// TwinCAT 3 PLC project LoadPCBAProject
// ProgramVersion: 3.1.4023.0
// libraries:
//   GreatechTemplate, * (Greatech)
//   Tc2_Standard, * (Beckhoff Automation GmbH)
//   Tc2_System, * (Beckhoff Automation GmbH)
//   Tc2_Utilities, * (Beckhoff Automation GmbH)
//   Tc3_Module, * (Beckhoff Automation GmbH)
// project tree:
//   DUTs/ ST_BarcodeScanner.TcDUT, ST_ModulePerformance.TcDUT, ST_OEETime.TcDUT, ST_Position.TcDUT, ST_ScaraCurrentPos.TcDUT, ST_ScaraRobot.TcDUT, ST_ScaraRobotCmd.TcDUT, ST_VisionRecipe.TcDUT
//   GVLs/ DeviceMapping.TcGVL, G_Auto.TcGVL, G_Error.TcGVL, G_Home.TcGVL, G_IO.TcGVL, G_MachineControl.TcGVL, G_Manual.TcGVL, G_Recipe.TcGVL, G_Robot.TcGVL, G_Safety.TcGVL, G_Scanner.TcGVL, G_Values.TcGVL, G_Vision.TcGVL
//   / PlcTask.TcTTO
//   POUs/Function Block/ FB_CognexBarcodeScanner.TcPOU, FB_OEETime.TcPOU, FB_RealToBytes.TcPOU
//   POUs/Function/ F_BytesToWord.TcPOU, F_ReadRobotPosition.TcPOU
//   POUs/General/ DoorLock.TcPOU, ErrorHandle.TcPOU, Initialize.TcPOU, MAIN.TcPOU, NewLotEndLot.TcPOU
//   POUs/General/Mapping/ Mapping_EIP.TcPOU, Mapping_IO.TcPOU
//   POUs/ POU_TestGitHub.TcPOU
//   POUs/Station/ST00_Conveyor/ ST00_ChangeRecipe.TcPOU, ST00_Cylinder.TcPOU, ST00_Sequence.TcPOU
//   POUs/Station/ST10_BarcodeScanner/ ST10_BarcodeScanner.TcPOU, ST10_Sequence.TcPOU
//   POUs/Station/ST20_PickNPlace/Robot/ ST20_RobotManualControl.TcPOU, ST20_RobotSequence.TcPOU, ST20_VisionManualControl.TcPOU
//   POUs/Station/ST20_PickNPlace/ ST20_ChangeRecipe.TcPOU, ST20_Home.TcPOU, ST20_Sequence.TcPOU
//   POUs/Station/ST20_PickNPlace/TrayLoader/ ST20_TraySequence.TcPOU, ST20_BarcodeScanner.TcPOU
// real-time tasks:
//   TASK PlcTask: cycle T#10ms, priority 20, ADS port 350

CONFIGURATION LoadPCBAProject
    RESOURCE PLC ON TwinCAT3
        TASK PlcTask(INTERVAL := T#10ms, PRIORITY := 20);
        PROGRAM MAIN WITH PlcTask : MAIN;
    END_RESOURCE
END_CONFIGURATION

// ---- DUTs/ST_BarcodeScanner.TcDUT
TYPE ST_BarcodeScanner :
STRUCT
	In_TriggerReady			: BOOL;
	In_TriggerAck			: BOOL;
	In_Acquiring			: BOOL;
	In_MissedAcq			: BOOL;
	In_noname0_arrBIT_0		: BOOL;
	In_noname0_arrBIT_1		: BOOL;
	In_noname0_arrBIT_2		: BOOL;
	In_noname0_arrBIT_3		: BOOL;
	In_Decoding				: BOOL;
	In_DecodeComplete		: BOOL;
	In_ResultsBufferOverrun : BOOL;
	In_ResultAvailable		: BOOL;
	In_noname1_arrBIT_0		: BOOL;
	In_noname1_arrBIT_1		: BOOL;
	In_noname1_arrBIT_2		: BOOL;
	In_GeneralFault			: BOOL;
	In_SoftEventAck0		: BOOL;
	In_SoftEventAck1		: BOOL;
	In_SoftEventAck2		: BOOL;
	In_SoftEventAck3		: BOOL;
	In_SoftEventAck4		: BOOL;
	In_SoftEventAck5		: BOOL;
	In_SoftEventAck6		: BOOL;
	In_SoftEventAck7		: BOOL;
	In_noname2_arrBYTE_0	: BYTE;
	In_noname2_arrBYTE_1	: BYTE;
	In_noname2_arrBYTE_2	: BYTE;
	In_TriggerID			: UINT;
	In_ResultID				: UINT;
	In_ResultCode			: UINT;
	In_ResultExtended		: UINT;
	In_ResultLength			: UINT;
	In_ResultData			: ARRAY [0..479] OF BYTE;
	
	
	Out_TriggerEnable		: BOOL;
	Out_Trigger				: BOOL;
	Out_BufferResultsEnable	: BOOL;
	Out_ResultAck			: BOOL;
	Out_noname0_arrBIT_0	: BOOL;
	Out_noname0_arrBIT_1	: BOOL;
	Out_noname0_arrBIT_2	: BOOL;
	Out_noname0_arrBIT_3	: BOOL;
	Out_SoftEvent0			: BOOL;
	Out_SoftEvent1			: BOOL;
	Out_SoftEvent2			: BOOL;
	Out_SoftEvent3			: BOOL;
	Out_SoftEvent4			: BOOL;
	Out_SoftEvent5			: BOOL;
	Out_SoftEvent6			: BOOL;
	Out_SoftEvent7			: BOOL;
	Out_noname1_arrBYTE_0	: BYTE;
	Out_noname1_arrBYTE_1	: BYTE;
	Out_UserDataOption		: UINT;
	Out_UserDataLength		: UINT;
	Out_UserData			: ARRAY [0..487] OF BYTE;
END_STRUCT
END_TYPE

// ---- DUTs/ST_ModulePerformance.TcDUT
TYPE ST_ModulePerformance :
STRUCT
	tBoardArrivalTime 	: TIME;
	tBoardLiftUpTime	: TIME;
	tPalletToFlipperTime: TIME;
	tFlippingTime		: TIME;
	tFlipperToPalletTime: TIME;
	tBoardLiftDownTime	: TIME;
	tBoardLeaveTime		: TIME;
	tMESResponseTime	: TIME;
END_STRUCT
END_TYPE

// ---- DUTs/ST_OEETime.TcDUT
TYPE ST_OEETime :
STRUCT
	RunTime		: LTIME;
	IdleTime 	: LTIME;
	DownTime	: LTIME;
END_STRUCT
END_TYPE

// ---- DUTs/ST_Position.TcDUT
TYPE ST_Position :
STRUCT
	Xpos: REAL;
	Ypos: REAL;
	Zpos: REAL;
	Apos: REAL;
END_STRUCT
END_TYPE

// ---- DUTs/ST_ScaraCurrentPos.TcDUT
TYPE ST_ScaraCurrentPos :
STRUCT
	RobotCurrentPos_X : REAL;
	RobotCurrentPos_Y : REAL;
	RobotCurrentPos_Z : REAL;
	RobotCurrentPos_A : REAL;
END_STRUCT
END_TYPE

// ---- DUTs/ST_ScaraRobot.TcDUT
TYPE ST_ScaraRobot :
STRUCT
	//Robot to PLC
	bReady				: BOOL; 
	bRunning		 	: BOOL; 
	bPaused			 	: BOOL; 
	bStopped		 	: BOOL; 
	bError			 	: BOOL; 
	bSafeguardON	 	: BOOL; 
	bEstopON		 	: BOOL; 
	bSerror			 	: BOOL; 
	bWarning 		 	: BOOL; 
	bEnabled		 	: BOOL; 
	bAcknowledged	 	: BOOL; 
	bHomeDone 			: BOOL;	
	bStandbyPositionDone: BOOL; 
	bClearMessageDone	: BOOL; 

	//PLC to Robot              
	bStop			 	: BOOL; 
	bStart			 	: BOOL; 
	bPause			 	: BOOL; 
	bContinue		 	: BOOL; 
	bReset 			 	: BOOL; 
	bEnable 		 	: BOOL; 
	bAppID0 		 	: BOOL; 
	bAppID1 		 	: BOOL; 
	bAppID2 		 	: BOOL; 
	bAcknowledgeMsg	 	: BOOL; 
	bHome 				: BOOL; 
	bStandbyPosition 	: BOOL; 
	bClearMessage		: BOOL; 
      
	wOutLowerX			: WORD; //byte 5 and 6
	wOutUpperX			: WORD; //byte 7 and 8
	wOutLowerY			: WORD; //byte 9 and 10
	wOutUpperY			: WORD; //byte 11 and 12
	wOutLowerZ			: WORD; //byte 13 and 14
	wOutUpperZ			: WORD; //byte 15 and 16
	wOutLowerA			: WORD; //byte 17 and 18
	wOutUpperA			: WORD; //byte 19 and 20
	
END_STRUCT
END_TYPE

// ---- DUTs/ST_ScaraRobotCmd.TcDUT
TYPE ST_ScaraRobotCmd :
STRUCT
//===================================
//Output
//===================================

	bRobotPalletFiducial1				: BOOL;
	bRobotPalletFiducial2				: BOOL;
	bRobotTrayFiducial1					: BOOL;
	bRobotTrayFiducial2					: BOOL;
	bRobotPickPCBA						: BOOL;
	bRobotPlacePCBA						: BOOL;
	bRobotStandbyAtPallet				: BOOL;
	bRobotStandbyAtTray					: BOOL;
	
	bRobotGripperOnOff					: BOOL;
	
	bRobotCheckDatum					: BOOL;
	
	bRobotDryRun						: BOOL;

//===================================
//Input
//===================================
	
	bRobotPalletFiducial1Done			: BOOL;
	bRobotPalletFiducial2Done			: BOOL;
	bRobotTrayFiducial1Done				: BOOL;
	bRobotTrayFiducial2Done				: BOOL;
	bRobotPickPCBADone					: BOOL;
	bRobotPlacePCBADone					: BOOL;
	bRobotStandbyAtPalletDone			: BOOL;
	bRobotStandbyAtTrayDone				: BOOL;
	
	bRobotGripperOnDone					: BOOL;
	
	bRobotCheckDatumDone				: BOOL;
	
	bRobotFailPlaceOverPress			: BOOL;

	//PLC to Robot
	rRobotPlace_X						: REAL;
	rRobotPlace_Y						: REAL;
	rRobotPlace_Z 						: REAL;
	rRobotPlace_A						: REAL;
	
END_STRUCT
END_TYPE

// ---- DUTs/ST_VisionRecipe.TcDUT
TYPE ST_VisionRecipe :
STRUCT
	stFiducialDistance2Value: ST_Position;
	stPocket : ST_Position;
END_STRUCT
END_TYPE

// ---- GVLs/DeviceMapping.TcGVL
{attribute 'qualified_only'}
VAR_GLOBAL
//===========================================================	
// IO
//===========================================================
	Input00_00		AT %I*	: BOOL;
	Input00_01		AT %I*	: BOOL;
	Input00_02		AT %I*	: BOOL;
	Input00_03		AT %I*	: BOOL;
	Input00_04		AT %I*	: BOOL;
	Input00_05		AT %I*	: BOOL;
	Input00_06		AT %I*	: BOOL;
	Input00_07		AT %I*	: BOOL;
	Input00_08		AT %I*	: BOOL;
	Input00_09		AT %I*	: BOOL;
	Input00_10		AT %I*	: BOOL;
	Input00_11		AT %I*	: BOOL;
	Input00_12		AT %I*	: BOOL;
	Input00_13		AT %I*	: BOOL;
	Input00_14		AT %I*	: BOOL;
	Input00_15		AT %I*	: BOOL;
	
	Input01_00		AT %I*	: BOOL;
	Input01_01		AT %I*	: BOOL;
	Input01_02		AT %I*	: BOOL;
	Input01_03		AT %I*	: BOOL;
	Input01_04		AT %I*	: BOOL;
	Input01_05		AT %I*	: BOOL;
	Input01_06		AT %I*	: BOOL;
	Input01_07		AT %I*	: BOOL;
	Input01_08		AT %I*	: BOOL;
	Input01_09		AT %I*	: BOOL;
	Input01_10		AT %I*	: BOOL;
	Input01_11		AT %I*	: BOOL;
	Input01_12		AT %I*	: BOOL;
	Input01_13		AT %I*	: BOOL;
	Input01_14		AT %I*	: BOOL;
	Input01_15		AT %I*	: BOOL;
	
	Input02_00		AT %I*	: BOOL;
	Input02_01		AT %I*	: BOOL;
	Input02_02		AT %I*	: BOOL;
	Input02_03		AT %I*	: BOOL;
	Input02_04		AT %I*	: BOOL;
	Input02_05		AT %I*	: BOOL;
	Input02_06		AT %I*	: BOOL;
	Input02_07		AT %I*	: BOOL;
	Input02_08		AT %I*	: BOOL;
	Input02_09		AT %I*	: BOOL;
	Input02_10		AT %I*	: BOOL;
	Input02_11		AT %I*	: BOOL;
	Input02_12		AT %I*	: BOOL;
	Input02_13		AT %I*	: BOOL;
	Input02_14		AT %I*	: BOOL;
	Input02_15		AT %I*	: BOOL;
	
	
	Output00_00		AT %Q*	: BOOL;
	Output00_01		AT %Q*	: BOOL;
	Output00_02		AT %Q*	: BOOL;
	Output00_03		AT %Q*	: BOOL;
	Output00_04		AT %Q*	: BOOL;
	Output00_05		AT %Q*	: BOOL;
	Output00_06		AT %Q*	: BOOL;
	Output00_07		AT %Q*	: BOOL;
	Output00_08		AT %Q*	: BOOL;
	Output00_09		AT %Q*	: BOOL;
	Output00_10		AT %Q*	: BOOL;
	Output00_11		AT %Q*	: BOOL;
	Output00_12		AT %Q*	: BOOL;
	Output00_13		AT %Q*	: BOOL;
	Output00_14		AT %Q*	: BOOL;
	Output00_15		AT %Q*	: BOOL;
	
	Output01_00		AT %Q*	: BOOL;
	Output01_01		AT %Q*	: BOOL;
	Output01_02		AT %Q*	: BOOL;
	Output01_03		AT %Q*	: BOOL;
	Output01_04		AT %Q*	: BOOL;
	Output01_05		AT %Q*	: BOOL;
	Output01_06		AT %Q*	: BOOL;
	Output01_07		AT %Q*	: BOOL;
	Output01_08		AT %Q*	: BOOL;
	Output01_09		AT %Q*	: BOOL;
	Output01_10		AT %Q*	: BOOL;
	Output01_11		AT %Q*	: BOOL;
	Output01_12		AT %Q*	: BOOL;
	Output01_13		AT %Q*	: BOOL;
	Output01_14		AT %Q*	: BOOL;
	Output01_15		AT %Q*	: BOOL;
	
	Output02_00		AT %Q*	: BOOL;
	Output02_01		AT %Q*	: BOOL;
	Output02_02		AT %Q*	: BOOL;
	Output02_03		AT %Q*	: BOOL;
	Output02_04		AT %Q*	: BOOL;
	Output02_05		AT %Q*	: BOOL;
	Output02_06		AT %Q*	: BOOL;
	Output02_07		AT %Q*	: BOOL;
	Output02_08		AT %Q*	: BOOL;
	Output02_09		AT %Q*	: BOOL;
	Output02_10		AT %Q*	: BOOL;
	Output02_11		AT %Q*	: BOOL;
	Output02_12		AT %Q*	: BOOL;
	Output02_13		AT %Q*	: BOOL;
	Output02_14		AT %Q*	: BOOL;
	Output02_15		AT %Q*	: BOOL;
	
//===========================================================	
// Safety IO
//===========================================================
	SafetyInput01_01		AT %I*	: BOOL;
	SafetyInput01_02		AT %I*	: BOOL;
	SafetyInput01_03		AT %I*	: BOOL;
	SafetyInput01_04		AT %I*	: BOOL;
	SafetyInput01_05		AT %I*	: BOOL;
	SafetyInput01_06		AT %I*	: BOOL;
	SafetyInput01_07		AT %I*	: BOOL;
	SafetyInput01_08		AT %I*	: BOOL;

	SafetyOutput01_01		AT %Q*	: BOOL;
	SafetyOutput01_02		AT %Q*	: BOOL;
	SafetyOutput01_03		AT %Q*	: BOOL;
	SafetyOutput01_04		AT %Q*	: BOOL;
	SafetyOutput01_05		AT %Q*	: BOOL;
	SafetyOutput01_06		AT %Q*	: BOOL;
	SafetyOutput01_07		AT %Q*	: BOOL;
	SafetyOutput01_08		AT %Q*	: BOOL;
	

//===========================================================	
// EIP
//===========================================================
// Robot
	KUKA_To_PLC		AT %I* 	: ARRAY[1..128] OF BYTE;
	PLC_To_KUKA		AT %Q*	: ARRAY[1..128] OF BYTE;
	
	
//Barcode Scanner
	BarcodeScanner_To_PLC 	AT %I* 	:  ST_BarcodeScanner;
	PLC_To_BarcodeScanner 	AT %Q* 	:  ST_BarcodeScanner;
	
	
END_VAR

// ---- GVLs/G_Auto.TcGVL
{attribute 'qualified_only'}
VAR_GLOBAL
//===================================
//General
//===================================	
	A_bOverallStationStatus				: BOOL; //TO CONVEYOR INCOMING A_BSTATION FAILED FALSE, JOB DONE FALSE ( trigger HMI to collect data wait HMI false)
	A_bUpdatedMESStationStatus			: BOOL; // decide whether true: pass false: failed //
	//Pallet serial number eg: 12344
	//
	
//===================================
//Conveyor
//===================================
	A00_bLifterCylUp			: BOOL;
	A00_bLifterCylUpDone		: BOOL;
	A00_bLifterCylDown			: BOOL;
	A00_bLifterCylDownDone		: BOOL;
                            	
	A00_bStopperCylBlock		: BOOL;
	A00_bStopperCylBlockDone	: BOOL;	
	A00_bStopperCylRelease		: BOOL;
	A00_bStopperCylReleaseDone	: BOOL;	

	
//===================================
//ST10 Barcode Scanner
//===================================
	A10_bTriggerScannerEnable		: BOOL;
	A10_bTriggerScannerEnableReady 	: BOOL;
	A10_bTriggerScanner				: BOOL;
	A10_bTriggerScannerDone			: BOOL;
	A10_bScannerResultDone			: BOOL;
	A10_sScannerBarcode				: STRING;

//===================================
//ST20 Pick And Place
//===================================	
	A20_bMESCheckDone				: BOOL;
	A20_bMESPass					: BOOL;
	A20_bMESCheck					: BOOL;
	
	A20_bTriggerScannerEnable		: BOOL;
	A20_bTriggerScannerEnableReady 	: BOOL;
	A20_bTriggerScanner				: BOOL;
	A20_bTriggerScannerDone			: BOOL;
	A20_bScannerResultDone			: BOOL;
	A20_sScannerBarcode				: STRING;
	
	A20_bIsNewTray					: BOOL;
	A20_bTrayReady					: BOOL;
	A20_bTrayFinish					: BOOL;
	
	A20_bRobotInitialize			: BOOL;
	A20_bRobotInitializeDone		: BOOL;
	A20_bPalletReady				: BOOL;
	                            	
	A20_bRobotAtStandbyTray			: BOOL;
	A20_bRobotAtStandbyPallet		: BOOL;
	                            	
	//Robot                     	
	A20_bRobotChangeRecipe			: BOOL;
	A20_bRobotChangeRecipeDone		: BOOL;
	
	A20_bRobotCheckDatum			: BOOL;
	A20_bRobotCheckDatumDone		: BOOL;

END_VAR

// ---- GVLs/G_Error.TcGVL
{attribute 'qualified_only'}
VAR_GLOBAL
//===================================
//Machine Control MD1000 - MD1004
//===================================	

	E_EmgStop							AT %MX4000.0 :BOOL;
	
//===================================
//Warning MD1005 - MD1007
//===================================	
	

//===================================
//Conveyor MD1008 - MD1009
//===================================
	E00_LifterCylUp 					AT %MX4032.0: BOOL;
	E00_LifterCylDown 					AT %MX4032.1: BOOL;
	                        		
	E00_StopperCylBlock					AT %MX4032.2: BOOL;
	E00_StopperCylRelease				AT %MX4032.3: BOOL;
	

//===================================
//ST10 Barcode Scanner MD1010
//===================================
	E10_BarcodeScannerDeviceError		AT %MX4040.0: BOOL;
	E10_BarcodeTimeout					AT %MX4040.1: BOOL;
	
	
//===================================
//ST20 Pick And Place MD1020
//===================================
	
	E20_BarcodeScannerDeviceError			AT %MX4080.0: BOOL;
	E20_BarcodeTimeout						AT %MX4080.1: BOOL;
	
	E20_VisionTimeOutInspection				AT %MX4081.0: BOOL;

	E20_RobotFailHome 						AT %MX4082.0: BOOL;
	E20_RobotFailStart			        	AT %MX4082.1: BOOL;
	E20_RobotFailServoOn		        	AT %MX4082.2: BOOL;
    E20_RobotFailToInitialize	        	AT %MX4082.3: BOOL;
	E20_RobotFailGetID						AT %MX4082.4: BOOL;

	E20_RobotTimeOutFailToPalletFiducial_1	AT %MX4083.0: BOOL;
	E20_RobotTimeOutFailToPalletFiducial_2	AT %MX4083.1: BOOL;
	E20_RobotTimeOutFailToTrayFiducial_1	AT %MX4083.2: BOOL;
	E20_RobotTimeOutFailToTrayFiducial_2	AT %MX4083.3: BOOL;
	E20_RobotTimeOutFailToPickPCBA			AT %MX4083.4: BOOL;
	E20_RobotTimeOutFailToPlacePCBA			AT %MX4083.5: BOOL;
	E20_RobotTimeOutFailToStandbyPallet		AT %MX4083.6: BOOL;
	E20_RobotTimeOutFailToStandbyTray		AT %MX4083.7: BOOL;
	
	E20_RobotFailDatumPos					AT %MX4084.0: BOOL;
	E20_VisionTimeOutDatumCheck				AT %MX4084.1: BOOL;
	E20_RobotFailPlaceOverpress				AT %MX4084.2: BOOL;
END_VAR

// ---- GVLs/G_Home.TcGVL
{attribute 'qualified_only'}
VAR_GLOBAL
	
//===================================
//Conveyor
//===================================
	H00_bLifterCylUp			: BOOL;
	H00_bLifterCylUpDone		: BOOL;
	H00_bLifterCylDown			: BOOL;
	H00_bLifterCylDownDone		: BOOL;

	H00_bStopperCylBlock		: BOOL;
	H00_bStopperCylBlockDone	: BOOL;	
	H00_bStopperCylRelease		: BOOL;
	H00_bStopperCylReleaseDone	: BOOL;	

//===================================
//ST10 Barcode Scanner
//===================================
	
//===================================
//ST20 Pick And Place
//===================================
	H20_bHome 					: BOOL;
	H20_bHomeDone				: BOOL;


END_VAR

// ---- GVLs/G_IO.TcGVL
{attribute 'qualified_only'}
VAR_GLOBAL
	
//===================================
//Input
//===================================

	I_StartPushButton 		: BOOL;
	I_ResetPushButton 		: BOOL;
	I_StopPushButton 		: BOOL;
	I_LifterUp				: BOOL;
	I_LifterDown			: BOOL;

//===================================
//Output
//===================================
	O_StartPushButton		: BOOL;
	O_ResetPushButton	 	: BOOL;
	O_StopPushButton 		: BOOL;
	O_LifterUp				: BOOL;
	O_LifterDown			: BOOL;
	
//===================================
//Safety Input
//===================================
 
	SI_FrontRightEmoCH1_1 						: BOOL;
	SI_FrontRightEmoCH1_2 						: BOOL;
	SI_FrontLeftEmoCH1_1 						: BOOL;
	SI_FrontLeftEmoCH1_2						: BOOL;
	SI_FrontRightEmoCH2_1						: BOOL;
	SI_FrontRightEmoCH2_2						: BOOL;
	SI_FrontLeftEmoCH2_1						: BOOL;
	SI_FrontLeftEmoCH2_2						: BOOL;
	
//===================================
//Safety Output
//===================================
	SO_CutOffContratorAcPower_1					: BOOL;
	SO_CutOffContratorAcPower_2 				: BOOL;
	SO_STO2_1 									: BOOL;
	SO_STO2_2									: BOOL;
	SO_STO1_1									: BOOL;
	SO_STO1_2									: BOOL;
	SO_Robot1_Acknowledge_1						: BOOL;
	SO_Robot1_Acknowledge_2						: BOOL;
	
END_VAR

// ---- GVLs/G_MachineControl.TcGVL
{attribute 'qualified_only'}
VAR_GLOBAL CONSTANT
	iStation				: INT := 2;
END_VAR

VAR_GLOBAL
	stMachineOperateMode	:ST_MachineOperateMode;
	stMachineCurrentMode	:ST_MachineCurrentMode;
	stOEETime				:ST_OEETime;
	arrstStationControl		:ARRAY[0..iStation] OF ST_StationStructure;
	arrsStationCycleTime	:ARRAY[0..iStation] OF STRING;
	
	bMainError				:BOOL;
	bMachineReset			:BOOL;
	bInitialize				:BOOL;
	bInitializeDone			:BOOL;
	bDryRun					:BOOL;
	bDoorIsLocked			:BOOL;
	bBypassDoor				:BOOL;
	
	bSafetyEnable			:BOOL;
	
	bBypassMES				: BOOL;
	bBypassWholeMachine		: BOOL;
	
	sMachineStatus			:STRING;
	sMachineCurrentStatus	:STRING;
	
	arrsST10StepStatus	: ARRAY [1..100] OF STRING;
	arrtimeST10StepTime	: ARRAY [1..100] OF TIME;
	
	arrsST20StepStatus	: ARRAY [1..100] OF STRING;
	arrtimeST20StepTime	: ARRAY [1..100] OF TIME;
	
	//
END_VAR

// ---- GVLs/G_Manual.TcGVL
{attribute 'qualified_only'}
VAR_GLOBAL
//===================================
//General
//===================================
	M_bNewLot					: BOOL;
	M_bNewLotConfirm			: BOOL;
	M_bLotStarted				: BOOL;
	M_bEndLot					: BOOL;
	M_bDoorLock					: BOOL;
	M_bLoadRecipe				: BOOL;
 
	M_bStart					: BOOL;
	M_bStop						: BOOL;
	M_bReset					: BOOL;
//===================================
//Machine Control
//===================================
	M_CheckIOUse				: BOOL;
	
//===================================
//Conveyor
//===================================

	M00_bLifterCylUp			: BOOL;
	M00_bLifterCylUpDone		: BOOL;
	M00_bLifterCylDown			: BOOL;
	M00_bLifterCylDownDone		: BOOL;
	
	M00_bStopperCylBlock		: BOOL;
	M00_bStopperCylBlockDone	: BOOL;	
	M00_bStopperCylRelease		: BOOL;
	M00_bStopperCylReleaseDone	: BOOL;	
	
	
//===================================
//ST10 Barcode Scanner
//===================================
	M10_bTriggerScannerEnable		: BOOL;
	M10_bTriggerScannerEnableReady 	: BOOL;
	M10_bTriggerScannerDone			: BOOL;
	M10_bTriggerScanner				: BOOL;
	M10_bScannerResultDone			: BOOL;
	M10_sScannerBarcode				: STRING;


//===================================
//ST20 Pick And Place
//===================================
	M20_bTriggerScannerEnable		: BOOL;
	M20_bTriggerScannerEnableReady 	: BOOL;
	M20_bTriggerScannerDone			: BOOL;
	M20_bTriggerScanner				: BOOL;
	M20_bScannerResultDone			: BOOL;
	M20_sScannerBarcode				: STRING;

	M20_bChangeRobotProgramID	: BOOL;
	M20_byteRobotProgramID		: BYTE;
	M20_bAppID0					: BOOL;
	M20_bAppID1					: BOOL;
	M20_bAppID2					: BOOL;
	
	M20_bRobotHome				: BOOL;
	M20_bRobotEnable			: BOOL;
	M20_bRobotStart				: BOOL;
	M20_bRobotStop				: BOOL;
	M20_bRobotReset				: BOOL;
	M20_bRobotPause				: BOOL;
	M20_bRobotContinue			: BOOL;
	M20_bRobotPowerOn			: BOOL;
	M20_bRobotStandbyPos		: BOOL;
	M20_bClearMessage			: BOOL;
	M20_bRobotGripperOnOff		: BOOL;
	M20_bRobotTrayFiducial1		: BOOL;
	M20_bRobotTrayFiducial2		: BOOL;
	M20_bRobotPalletFiducial1	: BOOL;
	M20_bRobotPalletFiducial2	: BOOL;
	M20_bRobotPickPCBAPos		: BOOL;
	M20_bRobotPlacePCBAPos		: BOOL;
	M20_bRobotAtStandbyTray		: BOOL;
	M20_bRobotAtStandbyPallet	: BOOL;
	M20_bWithVisionData			: BOOL;
	
	M20_bVisionTrayFiducial1	: BOOL;
	M20_bVisionTrayFiducial2	: BOOL;
	M20_bVisionPalletFiducial1	: BOOL;
	M20_bVisionPalletFiducial2	: BOOL;

END_VAR

// ---- GVLs/G_Recipe.TcGVL
{attribute 'qualified_only'}
VAR_GLOBAL
 
//===================================
// General 
//===================================
	R_sProductName					: STRING;
	
//===================================
//ST00 Conveyor
//===================================
//	R00_stConveyorWidthrecipe		: ST_WidthRecipe;
	
//===================================
//ST20 RobotSCARA
//===================================
	R20_byteRobotProgramID		: BYTE;
	R20_stTrayPosition			: ST_VisionRecipe;
	R20_rTrayZaxisPick			: REAL;
	R20_stPalletPosition		: ST_VisionRecipe;
	R20_rPalletZaxisPlace		: REAL;
END_VAR

// ---- GVLs/G_Robot.TcGVL
{attribute 'qualified_only'}
VAR_GLOBAL
	RobotKukaStandard : ST_ScaraRobot;
	RobotKukaCurrentPos : ST_ScaraCurrentPos;
	RobotKukaCmd : ST_ScaraRobotCmd;
END_VAR

// ---- GVLs/G_Safety.TcGVL
{attribute 'qualified_only'}
VAR_GLOBAL
END_VAR

// ---- GVLs/G_Scanner.TcGVL
{attribute 'qualified_only'}
VAR_GLOBAL
	//Scanner to PLC
	//Load Tray Scanner
	In_Signal_Tray			: ST_BarcodeScanner;
	Out_Signal_Tray			: ST_BarcodeScanner;
	
	
	//Load Tray Scanner
	In_Signal_Conveyor		: ST_BarcodeScanner;
	Out_Signal_Conveyor		: ST_BarcodeScanner;

END_VAR

// ---- GVLs/G_Values.TcGVL
{attribute 'qualified_only'}
VAR_GLOBAL
//===================================
//ST00 General 
//===================================
	VA_sProductName					: STRING;
	VA_iTotalReject					: INT;
	VA_iTotalPass					: INT;
	VA_iTotalInput					: INT;	
	VA_iTotalOutput					: INT;
//===================================
//ST00 Conveyor 
//===================================
	VA00_rConveyorWidth				: REAL;

//===================================
//ST20 RobotScara
//===================================
	VA20_byteRobotProgramID			: BYTE;	
	VA20_stTrayPosition				: ST_VisionRecipe;
	VA20_rTrayZaxisPick				: REAL;
	VA20_stPalletPosition			: ST_VisionRecipe;
	VA20_rPalletZaxisPlace			: REAL;
	VA20_sDatumVisionResultStatus	: STRING;
	VA20_stDatumVisionResultPos		: ST_Position;
	
END_VAR

// ---- GVLs/G_Vision.TcGVL
{attribute 'qualified_only'}
VAR_GLOBAL
	V20_sSendCmd				: STRING;
	V20_bTrigger				: BOOL;
	V20_bRespone				: BOOL;
	
	V20_stTrayPosition			: ST_VisionRecipe; //HMI to PLC to Vision
	V20_stResultTrayPosition	: ST_Position; //Vision to PLC to Robot
	
	V20_stPalletPosition		: ST_VisionRecipe; //HMI to PLC to Vision
	V20_stResultPalletPosition	: ST_Position; //Vision to PLC to Robot
	
	V20_sDatumVisionResultStatus	: STRING;
	V20_stDatumVisionResultPos		: ST_Position;
END_VAR

// ---- POUs/General/MAIN.TcPOU
PROGRAM MAIN_1
VAR
	fbTime : FB_LocalSystemTime := ( bEnable := TRUE, dwCycle := 1 );
	sTime: STRING;
	sDateTime: STRING;
	sDate: STRING;
	fbMachineControl: FB_MachineControl;
	bStationError: BOOL;
	bAllError: BOOL;
	fbOEETimer: FB_OEETime;
	RTIRIG_NewLot: R_TRIG;
END_VAR

fbTime();
POU_TestGitHub();
IF fbTime.bValid THEN
	sDateTime := DT_TO_STRING(SYSTEMTIME_TO_DT(fbTime.systemTime));
	sDate := MID(sDateTime,10,4);
	sTime := RIGHT(sDateTime,8);
END_IF

bStationError := G_MachineControl.arrstStationControl[0].bError OR G_MachineControl.arrstStationControl[1].bError OR G_MachineControl.arrstStationControl[2].bError;

bAllError := G_MachineControl.bMainError OR bStationError;

fbMachineControl(
	In_bAutoMode:= TRUE, 
	In_bManualMode:= , 
	In_bDryRunMode:= G_MachineControl.bDryRun, 
	IN_bStartButton:= , 
	IN_bStopButton:= , 
	IN_bResetButton:= , 
	IN_bEmergencyStop:= TRUE, 
	IN_bMainAirPressureSwitch:= TRUE, 
	In_bDoorLocked:= TRUE OR G_MachineControl.bDoorIsLocked OR G_MachineControl.bBypassDoor, 
	In_bSafetyModeON:= TRUE, 
	In_bSafetyModeOFF:= , 
	In_InitializeTimeout:= , 
	In_InitializeDone:= G_MachineControl.bInitializeDone,  
	In_bEndLot:= , 
	In_bError:= , 
	Out_bReset=> G_MachineControl.bMachineReset,  
	Out_bInitialize=> G_MachineControl.bInitialize, 
	Out_sCurrentState=> , 
	Out_bRunning=> , 
	Out_bErrorInitialize=> , 
	Out_bErrorDoorLock=> , 
	Out_bErrorSafety=> , 
	Out_bErrorEStop=> , 
	Out_bErrorSwitch=> , 
	Out_bErrorMainAirPressureSwitch=> , 
	Out_StartButtonLight=> , 
	Out_StopButtonLight=> , 
	Out_ResetButtonLight=> , 
	Out_RedTowerlight=> , 
	Out_YellowTowerlight=> , 
	Out_GreenTowerlight=> , 
	Out_BlueTowerlight=> , 
	Out_Buzzer=> , 
	InOut_OperateMode:= G_MachineControl.stMachineOperateMode, 
	InOut_CurrentMode:= G_MachineControl.stMachineCurrentMode);
	
IF G_MachineControl.bBypassWholeMachine THEN
	G_MachineControl.arrstStationControl[1].bByPassStation := TRUE;
	G_MachineControl.arrstStationControl[2].bByPassStation := TRUE;
END_IF
 
fbOEETimer(
	In_stMachineCurrentMode:= G_MachineControl.stMachineCurrentMode, 
	In_iTotalReject:= G_Values.VA_iTotalReject, 
	In_iTotalPass:= G_Values.VA_iTotalPass, 
	Out_iTotalOutput=> G_Values.VA_iTotalOutput, 
	InOut_stOEETime:= G_MachineControl.stOEETime);
 
RTIRIG_NewLot(CLK := G_Manual.M_bLotStarted); ///to do with conveyor
IF RTIRIG_NewLot.Q THEN
	G_MachineControl.stOEETime.IdleTime := LTIME#0MS;
	G_MachineControl.stOEETime.RunTime := LTIME#0MS;
	G_MachineControl.stOEETime.DownTime := LTime#0MS;
	G_Values.VA_iTotalReject := 0;
	G_Values.VA_iTotalPass := 0;
END_IF	
	
IF G_MachineControl.stMachineOperateMode.AUTO THEN
	G_MachineControl.sMachineStatus := 'Auto Mode';
ELSIF G_MachineControl.stMachineOperateMode.MANUAL THEN
	G_MachineControl.sMachineStatus := 'Manual Mode';
END_IF

IF G_MachineControl.stMachineCurrentMode.AUTO_RUNNING THEN
	G_MachineControl.sMachineCurrentStatus := 'Machine Running';
ELSIF G_MachineControl.stMachineCurrentMode.STOP THEN
	G_MachineControl.sMachineCurrentStatus := 'Machine Stopped';
ELSIF G_MachineControl.stMachineCurrentMode.INITIALIZE THEN
	G_MachineControl.sMachineCurrentStatus := 'Machine Initialize';	
ELSIF G_MachineControl.stMachineCurrentMode.ERROR_MODE THEN
	G_MachineControl.sMachineCurrentStatus := 'Machine Error';
ELSE
	G_MachineControl.sMachineCurrentStatus := '';
END_IF

IF G_MachineControl.stMachineOperateMode.DRYRUN THEN
	G_Robot.RobotKukaCmd.bRobotDryRun := TRUE;
ELSE
	G_Robot.RobotKukaCmd.bRobotDryRun := FALSE;
END_IF

Mapping_EIP();
Mapping_IO();
ErrorHandle();

ST00_ChangeRecipe();
ST00_Cylinder();
ST00_Sequence();

ST10_BarcodeScanner();
ST10_Sequence();

ST20_RobotManualControl();
ST20_RobotSequence();
ST20_BarcodeScanner();
ST20_TraySequence();
ST20_ChangeRecipe();
ST20_Home();
ST20_Sequence();

END_PROGRAM

// ---- POUs/Function Block/FB_OEETime.TcPOU
FUNCTION_BLOCK FB_OEETime
VAR_INPUT
	In_stMachineCurrentMode : ST_MachineCurrentMode;
	In_iTotalReject	: INT;
	In_iTotalPass	: INT;
END_VAR
VAR_OUTPUT
	Out_iTotalOutput	: INT;
END_VAR
VAR_IN_OUT
	InOut_stOEETime	: ST_OEETime;
END_VAR
VAR
	tonRunTimer			: ton;
	tonIdleTimer		: ton;
	tonDownTimer		: ton;
	tonUnknowTimer		: ton;
END_VAR

IF In_stMachineCurrentMode.AUTO_RUNNING THEN
	tonRunTimer(IN := In_stMachineCurrentMode.AUTO_RUNNING, PT:=T#1S);
	IF tonRunTimer.Q THEN
		tonRunTimer(IN := FALSE);
		InOut_stOEETime.RunTime := InOut_stOEETime.RunTime + TIME_TO_LTIME(tonRunTimer.PT);
	END_IF
ELSE
	InOut_stOEETime.RunTime := InOut_stOEETime.RunTime + TIME_TO_LTIME(tonRunTimer.ET);
	tonRunTimer(IN := FALSE);
END_IF

IF In_stMachineCurrentMode.STOP THEN
	tonIdleTimer(IN := In_stMachineCurrentMode.STOP, PT:=T#1S);
	IF tonIdleTimer.Q THEN
		tonIdleTimer(IN := FALSE);
		InOut_stOEETime.IdleTime := InOut_stOEETime.IdleTime + TIME_TO_LTIME(tonIdleTimer.PT);
	END_IF
ELSE
	InOut_stOEETime.IdleTime := InOut_stOEETime.IdleTime + TIME_TO_LTIME(tonIdleTimer.ET);
	tonIdleTimer(IN := FALSE);
END_IF

IF NOT In_stMachineCurrentMode.AUTO_RUNNING AND NOT In_stMachineCurrentMode.STOP AND NOT In_stMachineCurrentMode.DRYRUN_RUNNING
	AND NOT In_stMachineCurrentMode.INITIALIZE AND NOT In_stMachineCurrentMode.MANUAL_RUNNING AND NOT In_stMachineCurrentMode.ERROR_MODE THEN
	tonUnknowTimer(IN := TRUE, PT:=T#1S);
	IF tonUnknowTimer.Q THEN
		tonUnknowTimer(IN := FALSE);
		InOut_stOEETime.IdleTime := InOut_stOEETime.IdleTime + TIME_TO_LTIME(tonUnknowTimer.PT);
	END_IF
ELSE
	InOut_stOEETime.IdleTime := InOut_stOEETime.IdleTime + TIME_TO_LTIME(tonUnknowTimer.ET);
	tonUnknowTimer(IN := FALSE);
END_IF

IF In_stMachineCurrentMode.ERROR_MODE THEN
	tonDownTimer(IN := In_stMachineCurrentMode.ERROR_MODE, PT:=T#1S);
	IF tonDownTimer.Q THEN
		tonDownTimer(IN := FALSE);
		InOut_stOEETime.DownTime := InOut_stOEETime.DownTime + TIME_TO_LTIME(tonDownTimer.PT);
	END_IF
ELSE
	InOut_stOEETime.DownTime := InOut_stOEETime.DownTime + TIME_TO_LTIME(tonDownTimer.ET);
	tonDownTimer(IN := FALSE);
END_IF

Out_iTotalOutput := In_iTotalReject + In_iTotalPass;

END_FUNCTION_BLOCK

// ---- POUs/General/Initialize.TcPOU
PROGRAM Initialize
VAR
	Initialize_RTrig: R_TRIG;
	iStep : INT;
END_VAR

Initialize_RTrig(CLK:= G_MachineControl.bInitialize);
IF Initialize_RTrig.Q THEN
	G_MachineControl.bInitializeDone := FALSE;
	iStep := 10;
END_IF

CASE iStep OF
	10:
		//G_Home.H10_bHome := TRUE;
		G_Home.H20_bHome := TRUE;
		iStep := 20;
		
	20:
		IF G_Home.H20_bHomeDone THEN
			G_MachineControl.bInitialize := FALSE;
			G_MachineControl.bInitializeDone := TRUE;
			iStep := 0;
		END_IF
END_CASE

//Hello World

END_PROGRAM

// ---- POUs/POU_TestGitHub.TcPOU
PROGRAM POU_TestGitHub
VAR
	input : BOOL;
	output : BOOL;
END_VAR

output := input;

END_PROGRAM

// ---- POUs/General/Mapping/Mapping_EIP.TcPOU
PROGRAM Mapping_EIP
VAR
	fb_Place_PosX: FB_RealToBytes;
	fb_Place_PosY: FB_RealToBytes;
	fb_Place_PosZ: FB_RealToBytes;
	fb_Place_PosA: FB_RealToBytes;
END_VAR

//============================================================================================================
// PLC to Robot
//============================================================================================================
//Standard Byte 1 - 25
DeviceMapping.PLC_To_KUKA[1].0 := G_Robot.RobotKukaStandard.bStop; 			//Byte1.1//
DeviceMapping.PLC_To_KUKA[1].1 := G_Robot.RobotKukaStandard.bStart; 		//Byte1.2//
DeviceMapping.PLC_To_KUKA[1].2 := G_Robot.RobotKukaStandard.bPause;			//Byte1.3//
DeviceMapping.PLC_To_KUKA[1].3 := G_Robot.RobotKukaStandard.bContinue; 		//Byte1.4//
DeviceMapping.PLC_To_KUKA[1].4 := G_Robot.RobotKukaStandard.bReset; 		//Byte1.5//
DeviceMapping.PLC_To_KUKA[1].5 := G_Robot.RobotKukaStandard.bEnable; 		//Byte1.6//
DeviceMapping.PLC_To_KUKA[1].6 := G_Robot.RobotKukaStandard.bAppID0;		//Byte1.7//	
DeviceMapping.PLC_To_KUKA[1].7 := G_Robot.RobotKukaStandard.bAppID1;		//Byte1.8//	

DeviceMapping.PLC_To_KUKA[2].0 := G_Robot.RobotKukaStandard.bAppID2;			//Byte2.1//		
DeviceMapping.PLC_To_KUKA[2].1 := G_Robot.RobotKukaStandard.bAcknowledgeMsg;	//Byte2.2//
DeviceMapping.PLC_To_KUKA[2].2 := G_Robot.RobotKukaStandard.bHome;				//Byte2.3//
DeviceMapping.PLC_To_KUKA[2].3 := G_Robot.RobotKukaStandard.bStandbyPosition;	//Byte2.4//
DeviceMapping.PLC_To_KUKA[2].4 := G_Robot.RobotKukaStandard.bClearMessage;		//Byte2.5//

//PLC To robot Position 5 - 20 (Reserve)

fb_Place_PosX(
	IN_DATA:= G_Robot.RobotKukaCmd.rRobotPlace_X, 
	UpperByteA=> DeviceMapping.PLC_To_KUKA[5], 
	UpperByteB=> DeviceMapping.PLC_To_KUKA[6], 
	LowerByteC=> DeviceMapping.PLC_To_KUKA[7], 
	LowerByteD=> DeviceMapping.PLC_To_KUKA[8]);
	
fb_Place_PosY(
	IN_DATA:= G_Robot.RobotKukaCmd.rRobotPlace_Y, 
	UpperByteA=> DeviceMapping.PLC_To_KUKA[9], 
	UpperByteB=> DeviceMapping.PLC_To_KUKA[10], 
	LowerByteC=> DeviceMapping.PLC_To_KUKA[11], 
	LowerByteD=> DeviceMapping.PLC_To_KUKA[12]);
	
fb_Place_PosZ(
	IN_DATA:= G_Robot.RobotKukaCmd.rRobotPlace_Z, 
	UpperByteA=> DeviceMapping.PLC_To_KUKA[13], 
	UpperByteB=> DeviceMapping.PLC_To_KUKA[14], 
	LowerByteC=> DeviceMapping.PLC_To_KUKA[15], 
	LowerByteD=> DeviceMapping.PLC_To_KUKA[16]);
	
fb_Place_PosA(
	IN_DATA:= G_Robot.RobotKukaCmd.rRobotPlace_A, 
	UpperByteA=> DeviceMapping.PLC_To_KUKA[17], 
	UpperByteB=> DeviceMapping.PLC_To_KUKA[18], 
	LowerByteC=> DeviceMapping.PLC_To_KUKA[19], 
	LowerByteD=> DeviceMapping.PLC_To_KUKA[20]);
	
//Standard Command Byte 21 - 128	
DeviceMapping.PLC_To_KUKA[21].0 := G_Robot.RobotKukaCmd.bRobotPalletFiducial1;
DeviceMapping.PLC_To_KUKA[21].1 := G_Robot.RobotKukaCmd.bRobotPalletFiducial2;
DeviceMapping.PLC_To_KUKA[21].2 := G_Robot.RobotKukaCmd.bRobotTrayFiducial1;
DeviceMapping.PLC_To_KUKA[21].3 := G_Robot.RobotKukaCmd.bRobotTrayFiducial2;
DeviceMapping.PLC_To_KUKA[21].4 := G_Robot.RobotKukaCmd.bRobotPickPCBA;
DeviceMapping.PLC_To_KUKA[21].5 := G_Robot.RobotKukaCmd.bRobotPlacePCBA;
DeviceMapping.PLC_To_KUKA[21].6 := G_Robot.RobotKukaCmd.bRobotStandbyAtPallet;
DeviceMapping.PLC_To_KUKA[21].7 := G_Robot.RobotKukaCmd.bRobotStandbyAtTray;

DeviceMapping.PLC_To_KUKA[22].0 := G_Robot.RobotKukaCmd.bRobotGripperOnOff;
DeviceMapping.PLC_To_KUKA[22].1 := G_Robot.RobotKukaCmd.bRobotCheckDatum;
DeviceMapping.PLC_To_KUKA[22].2 := G_Robot.RobotKukaCmd.bRobotDryRun;

//============================================================================================================
// Robot to PLC
//============================================================================================================
//Standard Byte 1 - 25
G_Robot.RobotKukaStandard.bReady 				:= DeviceMapping.KUKA_To_PLC[1].0;  //Byte1.1//
G_Robot.RobotKukaStandard.bRunning 				:= DeviceMapping.KUKA_To_PLC[1].1;  //Byte1.2//
G_Robot.RobotKukaStandard.bPaused 				:= DeviceMapping.KUKA_To_PLC[1].2;  //Byte1.3//
G_Robot.RobotKukaStandard.bStopped 				:= DeviceMapping.KUKA_To_PLC[1].3;  //Byte1.4//
G_Robot.RobotKukaStandard.bError 				:= DeviceMapping.KUKA_To_PLC[1].4;  //Byte1.5// 
G_Robot.RobotKukaStandard.bSafeguardON 			:= DeviceMapping.KUKA_To_PLC[1].5;  //Byte1.6//
G_Robot.RobotKukaStandard.bEstopON 				:= DeviceMapping.KUKA_To_PLC[1].6;  //Byte1.7//
G_Robot.RobotKukaStandard.bSerror 				:= DeviceMapping.KUKA_To_PLC[1].7;  //Byte1.8//

G_Robot.RobotKukaStandard.bWarning				:= DeviceMapping.KUKA_To_PLC[2].0;  //Byte2.1//
G_Robot.RobotKukaStandard.bEnabled				:= DeviceMapping.KUKA_To_PLC[2].1;  //Byte2.2//
G_Robot.RobotKukaStandard.bAcknowledged			:= DeviceMapping.KUKA_To_PLC[2].2;  //Byte2.3//
G_Robot.RobotKukaStandard.bHomeDone				:= DeviceMapping.KUKA_To_PLC[2].3;  //Byte2.4//
G_Robot.RobotKukaStandard.bStandbyPositionDone	:= DeviceMapping.KUKA_To_PLC[2].4;  //Byte2.5

//Get Position - Start Byte 5 - 20
G_Robot.RobotKukaStandard.wOutUpperX			:= F_BytesToWord(IN_UpperByte:= DeviceMapping.KUKA_To_PLC[6], IN_LowerByte:= DeviceMapping.KUKA_To_PLC[5]);
G_Robot.RobotKukaStandard.wOutLowerX			:= F_BytesToWord(IN_UpperByte:= DeviceMapping.KUKA_To_PLC[8], IN_LowerByte:= DeviceMapping.KUKA_To_PLC[7]);
G_Robot.RobotKukaStandard.wOutUpperY			:= F_BytesToWord(IN_UpperByte:= DeviceMapping.KUKA_To_PLC[10], IN_LowerByte:= DeviceMapping.KUKA_To_PLC[9]);
G_Robot.RobotKukaStandard.wOutLowerY			:= F_BytesToWord(IN_UpperByte:= DeviceMapping.KUKA_To_PLC[12], IN_LowerByte:= DeviceMapping.KUKA_To_PLC[11]);
G_Robot.RobotKukaStandard.wOutUpperZ			:= F_BytesToWord(IN_UpperByte:= DeviceMapping.KUKA_To_PLC[14], IN_LowerByte:= DeviceMapping.KUKA_To_PLC[13]);
G_Robot.RobotKukaStandard.wOutLowerZ			:= F_BytesToWord(IN_UpperByte:= DeviceMapping.KUKA_To_PLC[16], IN_LowerByte:= DeviceMapping.KUKA_To_PLC[15]);
G_Robot.RobotKukaStandard.wOutUpperA			:= F_BytesToWord(IN_UpperByte:= DeviceMapping.KUKA_To_PLC[18], IN_LowerByte:= DeviceMapping.KUKA_To_PLC[17]);
G_Robot.RobotKukaStandard.wOutLowerA			:= F_BytesToWord(IN_UpperByte:= DeviceMapping.KUKA_To_PLC[20], IN_LowerByte:= DeviceMapping.KUKA_To_PLC[19]);

G_Robot.RobotKukaCurrentPos.RobotCurrentPos_X := F_ReadRobotPosition(IN_Upper:= G_Robot.RobotKukaStandard.wOutUpperX, IN_Lower:= G_Robot.RobotKukaStandard.wOutLowerX);
G_Robot.RobotKukaCurrentPos.RobotCurrentPos_Y := F_ReadRobotPosition(IN_Upper:= G_Robot.RobotKukaStandard.wOutUpperY, IN_Lower:= G_Robot.RobotKukaStandard.wOutLowerY);
G_Robot.RobotKukaCurrentPos.RobotCurrentPos_Z := F_ReadRobotPosition(IN_Upper:= G_Robot.RobotKukaStandard.wOutUpperZ, IN_Lower:= G_Robot.RobotKukaStandard.wOutLowerZ);
G_Robot.RobotKukaCurrentPos.RobotCurrentPos_A := F_ReadRobotPosition(IN_Upper:= G_Robot.RobotKukaStandard.wOutUpperA, IN_Lower:= G_Robot.RobotKukaStandard.wOutLowerA);

//Standard Command Byte 21 - 128
G_Robot.RobotKukaCmd.bRobotPalletFiducial1Done		:= DeviceMapping.KUKA_To_PLC[21].0;
G_Robot.RobotKukaCmd.bRobotPalletFiducial2Done		:= DeviceMapping.KUKA_To_PLC[21].1;
G_Robot.RobotKukaCmd.bRobotTrayFiducial1Done		:= DeviceMapping.KUKA_To_PLC[21].2;
G_Robot.RobotKukaCmd.bRobotTrayFiducial2Done		:= DeviceMapping.KUKA_To_PLC[21].3;
G_Robot.RobotKukaCmd.bRobotPickPCBADone				:= DeviceMapping.KUKA_To_PLC[21].4;
G_Robot.RobotKukaCmd.bRobotPlacePCBADone			:= DeviceMapping.KUKA_To_PLC[21].5;
G_Robot.RobotKukaCmd.bRobotStandbyAtPalletDone		:= DeviceMapping.KUKA_To_PLC[21].6;
G_Robot.RobotKukaCmd.bRobotStandbyAtTrayDone		:= DeviceMapping.KUKA_To_PLC[21].7;

G_Robot.RobotKukaCmd.bRobotGripperOnDone			:= DeviceMapping.KUKA_To_PLC[22].0;
G_Robot.RobotKukaCmd.bRobotCheckDatumDone			:= DeviceMapping.KUKA_To_PLC[22].1;
G_Robot.RobotKukaCmd.bRobotFailPlaceOverPress		:= DeviceMapping.KUKA_To_PLC[22].2;

//============================================================================================================
// Scanner Tray to PLC
//============================================================================================================
G_Scanner.In_Signal_Tray.In_TriggerReady		:= DeviceMapping.BarcodeScanner_To_PLC.In_TriggerReady;
G_Scanner.In_Signal_Tray.In_TriggerAck			:= DeviceMapping.BarcodeScanner_To_PLC.In_TriggerAck;
G_Scanner.In_Signal_Tray.In_Acquiring			:= DeviceMapping.BarcodeScanner_To_PLC.In_Acquiring;
G_Scanner.In_Signal_Tray.In_MissedAcq			:= DeviceMapping.BarcodeScanner_To_PLC.In_MissedAcq;	
G_Scanner.In_Signal_Tray.In_noname0_arrBIT_0 	:= DeviceMapping.BarcodeScanner_To_PLC.In_noname0_arrBIT_0;	
G_Scanner.In_Signal_Tray.In_noname0_arrBIT_1 	:= DeviceMapping.BarcodeScanner_To_PLC.In_noname0_arrBIT_1;
G_Scanner.In_Signal_Tray.In_noname0_arrBIT_2 	:= DeviceMapping.BarcodeScanner_To_PLC.In_noname0_arrBIT_2;
G_Scanner.In_Signal_Tray.In_noname0_arrBIT_3 	:= DeviceMapping.BarcodeScanner_To_PLC.In_noname0_arrBIT_3;	
G_Scanner.In_Signal_Tray.In_Decoding		 	:= DeviceMapping.BarcodeScanner_To_PLC.In_Decoding;
G_Scanner.In_Signal_Tray.In_DecodeComplete		:= DeviceMapping.BarcodeScanner_To_PLC.In_DecodeComplete;
G_Scanner.In_Signal_Tray.In_ResultsBufferOverrun:= DeviceMapping.BarcodeScanner_To_PLC.In_ResultsBufferOverrun;
G_Scanner.In_Signal_Tray.In_ResultAvailable		:= DeviceMapping.BarcodeScanner_To_PLC.In_ResultAvailable;
G_Scanner.In_Signal_Tray.In_noname1_arrBIT_0	:= DeviceMapping.BarcodeScanner_To_PLC.In_noname1_arrBIT_0;
G_Scanner.In_Signal_Tray.In_noname1_arrBIT_1	:= DeviceMapping.BarcodeScanner_To_PLC.In_noname1_arrBIT_1;
G_Scanner.In_Signal_Tray.In_noname1_arrBIT_2	:= DeviceMapping.BarcodeScanner_To_PLC.In_noname1_arrBIT_2;
G_Scanner.In_Signal_Tray.In_GeneralFault		:= DeviceMapping.BarcodeScanner_To_PLC.In_GeneralFault;
G_Scanner.In_Signal_Tray.In_SoftEventAck0		:= DeviceMapping.BarcodeScanner_To_PLC.In_SoftEventAck0;
G_Scanner.In_Signal_Tray.In_SoftEventAck1		:= DeviceMapping.BarcodeScanner_To_PLC.In_SoftEventAck1;
G_Scanner.In_Signal_Tray.In_SoftEventAck2		:= DeviceMapping.BarcodeScanner_To_PLC.In_SoftEventAck2;
G_Scanner.In_Signal_Tray.In_SoftEventAck3		:= DeviceMapping.BarcodeScanner_To_PLC.In_SoftEventAck3;
G_Scanner.In_Signal_Tray.In_SoftEventAck4		:= DeviceMapping.BarcodeScanner_To_PLC.In_SoftEventAck4;
G_Scanner.In_Signal_Tray.In_SoftEventAck5		:= DeviceMapping.BarcodeScanner_To_PLC.In_SoftEventAck5;
G_Scanner.In_Signal_Tray.In_SoftEventAck6		:= DeviceMapping.BarcodeScanner_To_PLC.In_SoftEventAck6;
G_Scanner.In_Signal_Tray.In_SoftEventAck7		:= DeviceMapping.BarcodeScanner_To_PLC.In_SoftEventAck7;
G_Scanner.In_Signal_Tray.In_noname2_arrBYTE_0	:= DeviceMapping.BarcodeScanner_To_PLC.In_noname2_arrBYTE_0;
G_Scanner.In_Signal_Tray.In_noname2_arrBYTE_1	:= DeviceMapping.BarcodeScanner_To_PLC.In_noname2_arrBYTE_1;
G_Scanner.In_Signal_Tray.In_noname2_arrBYTE_2	:= DeviceMapping.BarcodeScanner_To_PLC.In_noname2_arrBYTE_2;
G_Scanner.In_Signal_Tray.In_TriggerID			:= DeviceMapping.BarcodeScanner_To_PLC.In_TriggerID;
G_Scanner.In_Signal_Tray.In_ResultID			:= DeviceMapping.BarcodeScanner_To_PLC.In_ResultID;
G_Scanner.In_Signal_Tray.In_ResultCode			:= DeviceMapping.BarcodeScanner_To_PLC.In_ResultCode;
G_Scanner.In_Signal_Tray.In_ResultExtended		:= DeviceMapping.BarcodeScanner_To_PLC.In_ResultExtended;
G_Scanner.In_Signal_Tray.In_ResultLength		:= DeviceMapping.BarcodeScanner_To_PLC.In_ResultLength;
G_Scanner.In_Signal_Tray.In_ResultData			:= DeviceMapping.BarcodeScanner_To_PLC.In_ResultData;



//============================================================================================================
// PLC to Scanner Tray
//============================================================================================================
DeviceMapping.PLC_To_BarcodeScanner.Out_TriggerEnable 		:= G_Scanner.Out_Signal_Tray.Out_TriggerEnable;
DeviceMapping.PLC_To_BarcodeScanner.Out_Trigger 			:= G_Scanner.Out_Signal_Tray.Out_Trigger;
DeviceMapping.PLC_To_BarcodeScanner.Out_BufferResultsEnable	:= G_Scanner.Out_Signal_Tray.Out_BufferResultsEnable;
DeviceMapping.PLC_To_BarcodeScanner.Out_ResultAck	 		:= G_Scanner.Out_Signal_Tray.Out_ResultAck;
DeviceMapping.PLC_To_BarcodeScanner.Out_noname0_arrBIT_0 	:= G_Scanner.Out_Signal_Tray.Out_noname0_arrBIT_0;
DeviceMapping.PLC_To_BarcodeScanner.Out_noname0_arrBIT_1 	:= G_Scanner.Out_Signal_Tray.Out_noname0_arrBIT_1;
DeviceMapping.PLC_To_BarcodeScanner.Out_noname0_arrBIT_2 	:= G_Scanner.Out_Signal_Tray.Out_noname0_arrBIT_2;
DeviceMapping.PLC_To_BarcodeScanner.Out_noname0_arrBIT_3 	:= G_Scanner.Out_Signal_Tray.Out_noname0_arrBIT_3;
DeviceMapping.PLC_To_BarcodeScanner.Out_SoftEvent0	 		:= G_Scanner.Out_Signal_Tray.Out_SoftEvent0;
DeviceMapping.PLC_To_BarcodeScanner.Out_SoftEvent1	 		:= G_Scanner.Out_Signal_Tray.Out_SoftEvent1;
DeviceMapping.PLC_To_BarcodeScanner.Out_SoftEvent2	 		:= G_Scanner.Out_Signal_Tray.Out_SoftEvent2;
DeviceMapping.PLC_To_BarcodeScanner.Out_SoftEvent3	 		:= G_Scanner.Out_Signal_Tray.Out_SoftEvent3;
DeviceMapping.PLC_To_BarcodeScanner.Out_SoftEvent4	 		:= G_Scanner.Out_Signal_Tray.Out_SoftEvent4;
DeviceMapping.PLC_To_BarcodeScanner.Out_SoftEvent5	 		:= G_Scanner.Out_Signal_Tray.Out_SoftEvent5;
DeviceMapping.PLC_To_BarcodeScanner.Out_SoftEvent6	 		:= G_Scanner.Out_Signal_Tray.Out_SoftEvent6;
DeviceMapping.PLC_To_BarcodeScanner.Out_SoftEvent7	 		:= G_Scanner.Out_Signal_Tray.Out_SoftEvent7;
DeviceMapping.PLC_To_BarcodeScanner.Out_noname1_arrBYTE_0	:= G_Scanner.Out_Signal_Tray.Out_noname1_arrBYTE_0;
DeviceMapping.PLC_To_BarcodeScanner.Out_noname1_arrBYTE_1	:= G_Scanner.Out_Signal_Tray.Out_noname1_arrBYTE_1;
DeviceMapping.PLC_To_BarcodeScanner.Out_UserDataOption		:= G_Scanner.Out_Signal_Tray.Out_UserDataOption;
DeviceMapping.PLC_To_BarcodeScanner.Out_UserDataLength		:= G_Scanner.Out_Signal_Tray.Out_UserDataLength;
DeviceMapping.PLC_To_BarcodeScanner.Out_UserData			:= G_Scanner.Out_Signal_Tray.Out_UserData;


//============================================================================================================
// Scanner Conveyor to PLC
//============================================================================================================
G_Scanner.In_Signal_Conveyor.In_TriggerReady		:= DeviceMapping.BarcodeScanner_To_PLC.In_TriggerReady;
G_Scanner.In_Signal_Conveyor.In_TriggerAck			:= DeviceMapping.BarcodeScanner_To_PLC.In_TriggerAck;
G_Scanner.In_Signal_Conveyor.In_Acquiring			:= DeviceMapping.BarcodeScanner_To_PLC.In_Acquiring;
G_Scanner.In_Signal_Conveyor.In_MissedAcq			:= DeviceMapping.BarcodeScanner_To_PLC.In_MissedAcq;	
G_Scanner.In_Signal_Conveyor.In_noname0_arrBIT_0 	:= DeviceMapping.BarcodeScanner_To_PLC.In_noname0_arrBIT_0;	
G_Scanner.In_Signal_Conveyor.In_noname0_arrBIT_1 	:= DeviceMapping.BarcodeScanner_To_PLC.In_noname0_arrBIT_1;
G_Scanner.In_Signal_Conveyor.In_noname0_arrBIT_2 	:= DeviceMapping.BarcodeScanner_To_PLC.In_noname0_arrBIT_2;
G_Scanner.In_Signal_Conveyor.In_noname0_arrBIT_3 	:= DeviceMapping.BarcodeScanner_To_PLC.In_noname0_arrBIT_3;	
G_Scanner.In_Signal_Conveyor.In_Decoding		 	:= DeviceMapping.BarcodeScanner_To_PLC.In_Decoding;
G_Scanner.In_Signal_Conveyor.In_DecodeComplete		:= DeviceMapping.BarcodeScanner_To_PLC.In_DecodeComplete;
G_Scanner.In_Signal_Conveyor.In_ResultsBufferOverrun:= DeviceMapping.BarcodeScanner_To_PLC.In_ResultsBufferOverrun;
G_Scanner.In_Signal_Conveyor.In_ResultAvailable		:= DeviceMapping.BarcodeScanner_To_PLC.In_ResultAvailable;
G_Scanner.In_Signal_Conveyor.In_noname1_arrBIT_0	:= DeviceMapping.BarcodeScanner_To_PLC.In_noname1_arrBIT_0;
G_Scanner.In_Signal_Conveyor.In_noname1_arrBIT_1	:= DeviceMapping.BarcodeScanner_To_PLC.In_noname1_arrBIT_1;
G_Scanner.In_Signal_Conveyor.In_noname1_arrBIT_2	:= DeviceMapping.BarcodeScanner_To_PLC.In_noname1_arrBIT_2;
G_Scanner.In_Signal_Conveyor.In_GeneralFault		:= DeviceMapping.BarcodeScanner_To_PLC.In_GeneralFault;
G_Scanner.In_Signal_Conveyor.In_SoftEventAck0		:= DeviceMapping.BarcodeScanner_To_PLC.In_SoftEventAck0;
G_Scanner.In_Signal_Conveyor.In_SoftEventAck1		:= DeviceMapping.BarcodeScanner_To_PLC.In_SoftEventAck1;
G_Scanner.In_Signal_Conveyor.In_SoftEventAck2		:= DeviceMapping.BarcodeScanner_To_PLC.In_SoftEventAck2;
G_Scanner.In_Signal_Conveyor.In_SoftEventAck3		:= DeviceMapping.BarcodeScanner_To_PLC.In_SoftEventAck3;
G_Scanner.In_Signal_Conveyor.In_SoftEventAck4		:= DeviceMapping.BarcodeScanner_To_PLC.In_SoftEventAck4;
G_Scanner.In_Signal_Conveyor.In_SoftEventAck5		:= DeviceMapping.BarcodeScanner_To_PLC.In_SoftEventAck5;
G_Scanner.In_Signal_Conveyor.In_SoftEventAck6		:= DeviceMapping.BarcodeScanner_To_PLC.In_SoftEventAck6;
G_Scanner.In_Signal_Conveyor.In_SoftEventAck7		:= DeviceMapping.BarcodeScanner_To_PLC.In_SoftEventAck7;
G_Scanner.In_Signal_Conveyor.In_noname2_arrBYTE_0	:= DeviceMapping.BarcodeScanner_To_PLC.In_noname2_arrBYTE_0;
G_Scanner.In_Signal_Conveyor.In_noname2_arrBYTE_1	:= DeviceMapping.BarcodeScanner_To_PLC.In_noname2_arrBYTE_1;
G_Scanner.In_Signal_Conveyor.In_noname2_arrBYTE_2	:= DeviceMapping.BarcodeScanner_To_PLC.In_noname2_arrBYTE_2;
G_Scanner.In_Signal_Conveyor.In_TriggerID			:= DeviceMapping.BarcodeScanner_To_PLC.In_TriggerID;
G_Scanner.In_Signal_Conveyor.In_ResultID			:= DeviceMapping.BarcodeScanner_To_PLC.In_ResultID;
G_Scanner.In_Signal_Conveyor.In_ResultCode			:= DeviceMapping.BarcodeScanner_To_PLC.In_ResultCode;
G_Scanner.In_Signal_Conveyor.In_ResultExtended		:= DeviceMapping.BarcodeScanner_To_PLC.In_ResultExtended;
G_Scanner.In_Signal_Conveyor.In_ResultLength		:= DeviceMapping.BarcodeScanner_To_PLC.In_ResultLength;
G_Scanner.In_Signal_Conveyor.In_ResultData			:= DeviceMapping.BarcodeScanner_To_PLC.In_ResultData;



//============================================================================================================
// PLC to Scanner Conveyor
//============================================================================================================
DeviceMapping.PLC_To_BarcodeScanner.Out_TriggerEnable 		:= G_Scanner.Out_Signal_Conveyor.Out_TriggerEnable;
DeviceMapping.PLC_To_BarcodeScanner.Out_Trigger 			:= G_Scanner.Out_Signal_Conveyor.Out_Trigger;
DeviceMapping.PLC_To_BarcodeScanner.Out_BufferResultsEnable	:= G_Scanner.Out_Signal_Conveyor.Out_BufferResultsEnable;
DeviceMapping.PLC_To_BarcodeScanner.Out_ResultAck	 		:= G_Scanner.Out_Signal_Conveyor.Out_ResultAck;
DeviceMapping.PLC_To_BarcodeScanner.Out_noname0_arrBIT_0 	:= G_Scanner.Out_Signal_Conveyor.Out_noname0_arrBIT_0;
DeviceMapping.PLC_To_BarcodeScanner.Out_noname0_arrBIT_1 	:= G_Scanner.Out_Signal_Conveyor.Out_noname0_arrBIT_1;
DeviceMapping.PLC_To_BarcodeScanner.Out_noname0_arrBIT_2 	:= G_Scanner.Out_Signal_Conveyor.Out_noname0_arrBIT_2;
DeviceMapping.PLC_To_BarcodeScanner.Out_noname0_arrBIT_3 	:= G_Scanner.Out_Signal_Conveyor.Out_noname0_arrBIT_3;
DeviceMapping.PLC_To_BarcodeScanner.Out_SoftEvent0	 		:= G_Scanner.Out_Signal_Conveyor.Out_SoftEvent0;
DeviceMapping.PLC_To_BarcodeScanner.Out_SoftEvent1	 		:= G_Scanner.Out_Signal_Conveyor.Out_SoftEvent1;
DeviceMapping.PLC_To_BarcodeScanner.Out_SoftEvent2	 		:= G_Scanner.Out_Signal_Conveyor.Out_SoftEvent2;
DeviceMapping.PLC_To_BarcodeScanner.Out_SoftEvent3	 		:= G_Scanner.Out_Signal_Conveyor.Out_SoftEvent3;
DeviceMapping.PLC_To_BarcodeScanner.Out_SoftEvent4	 		:= G_Scanner.Out_Signal_Conveyor.Out_SoftEvent4;
DeviceMapping.PLC_To_BarcodeScanner.Out_SoftEvent5	 		:= G_Scanner.Out_Signal_Conveyor.Out_SoftEvent5;
DeviceMapping.PLC_To_BarcodeScanner.Out_SoftEvent6	 		:= G_Scanner.Out_Signal_Conveyor.Out_SoftEvent6;
DeviceMapping.PLC_To_BarcodeScanner.Out_SoftEvent7	 		:= G_Scanner.Out_Signal_Conveyor.Out_SoftEvent7;
DeviceMapping.PLC_To_BarcodeScanner.Out_noname1_arrBYTE_0	:= G_Scanner.Out_Signal_Conveyor.Out_noname1_arrBYTE_0;
DeviceMapping.PLC_To_BarcodeScanner.Out_noname1_arrBYTE_1	:= G_Scanner.Out_Signal_Conveyor.Out_noname1_arrBYTE_1;
DeviceMapping.PLC_To_BarcodeScanner.Out_UserDataOption		:= G_Scanner.Out_Signal_Conveyor.Out_UserDataOption;
DeviceMapping.PLC_To_BarcodeScanner.Out_UserDataLength		:= G_Scanner.Out_Signal_Conveyor.Out_UserDataLength;
DeviceMapping.PLC_To_BarcodeScanner.Out_UserData			:= G_Scanner.Out_Signal_Conveyor.Out_UserData;

END_PROGRAM

// ---- POUs/Function Block/FB_RealToBytes.TcPOU
FUNCTION_BLOCK FB_RealToBytes // Convert Real data into 4 bytes
VAR_INPUT
	IN_DATA : REAL; //The Input Data in Real Data type 
END_VAR
VAR_OUTPUT
	UpperByteA :BYTE; //  UpperByte 1 the 25-32 bits from the Data word (Count from Right) 
	UpperByteB :BYTE; //  UpperByte 2 the 17-24 bits from the Data word (Count from Right)
	LowerByteC :BYTE; //  LowerByte 1 the 9-16 bits from the Data word (Count from Right)
	LowerByteD :BYTE; //  LowerByte 2 the 1-8 bits from the Data word (Count from Right)
END_VAR
VAR
	b_Input : BYTE;
	w_Input : DWORD;
	r_Data 	: REAL;
	w_Input1: WORD;
	UpperDWord : DWORD;
	LowerDWord : DWORD;
	
	UpperWord: WORD;
	LowerWord: WORD;
	
	UpperWordA: WORD;
	UpperWordB: WORD;
	LowerWordA: WORD;
	LowerWordB: WORD;
END_VAR

r_Data :=  IN_DATA *1000; // remove decimal from real
w_Input:= TO_DWORD(r_Data);  // Change from real to word

// DWORD DATA Split into two DWORD 
UpperDWord := SHR(w_Input,16);
LowerDWord := w_Input - SHL(UpperDWord,16);

//  Change into WORD
UpperWord := TO_WORD(UpperDWord);
LowerWord := TO_WORD(LowerDWord);

// Convert WORD to Byte Calculation
UpperWordA := SHR(UpperWord,8);
UpperWordB := UpperWord - SHL(UpperWordA,8);

LowerWordA := SHR(LowerWord,8);
LowerWordB := LowerWord - SHL(LowerWordA,8);

//  Change into Byte
UpperByteA	:= TO_BYTE(UpperWordB);
UpperByteB	:= TO_BYTE(UpperWordA);

LowerByteC	:= TO_BYTE(LowerWordB);
LowerByteD	:= TO_BYTE(LowerWordA);

END_FUNCTION_BLOCK

// ---- POUs/Function/F_BytesToWord.TcPOU
FUNCTION F_BytesToWord : WORD // CONCAT two relative Bytes data into assending Order which Upper is bit 5-8 and Lower is bits 1-4
VAR_INPUT
	IN_UpperByte : BYTE; //The Upper 8 Bits data (1st Byte) from Full 16 Bits Data(WORD)
	IN_LowerByte : BYTE; //The Lower 8 Bits data (2st Byte) from Full 16 Bits Data(WORD)
END_VAR
VAR
	d_Input : WORD;
	i_Input : WORD;
END_VAR

// IN_UpperByte is Byte data from KUKA EIP
//d_Input = WORD
//INSERT WORD INTO DWORD
// SHL Shift Left 16 bit of data + Lower 16 bit of data 
// Convert DWORD to REAL 

d_Input :=  IN_UpperByte;
d_Input := SHL(d_Input,8) + IN_LowerByte;
F_BytesToWord:= TO_WORD(d_Input);

END_FUNCTION

// ---- POUs/Function/F_ReadRobotPosition.TcPOU
FUNCTION F_ReadRobotPosition : REAL
VAR_INPUT
	IN_Upper		: WORD; //The Upper 16 Bits data (1st WORD) from Full 32 Bits Data(DWORD)
	IN_Lower		: WORD; //The Lower 16 Bits data (2st WORD) from Full 32 Bits Data(DWORD)
END_VAR
VAR
	d_Input : DWORD;
	i_Input : REAL;
END_VAR

// IN_Upper is WORD from KUKA EIP
//d_Input = DWORD
//INSERT WORD INTO DWORD
// SHL Shift Left 16 bit of data + Lower 16 bit of data 
// Convert DWORD to REAL 

d_Input :=  IN_Upper;
d_Input := SHL(d_Input,16) + IN_Lower;
i_Input:= TO_REAL(DWORD_TO_DINT(d_Input));
F_ReadRobotPosition := (i_Input/1000);

END_FUNCTION

// ---- POUs/General/Mapping/Mapping_IO.TcPOU
PROGRAM Mapping_IO
VAR
END_VAR



G_IO.I_StartPushButton 				:= DeviceMapping.Input00_00;
G_IO.I_ResetPushButton 				:= DeviceMapping.Input00_01;
G_IO.I_StopPushButton 				:= DeviceMapping.Input00_02;






DeviceMapping.Output00_00 := G_IO.O_StartPushButton;
DeviceMapping.Output00_01 := G_IO.O_ResetPushButton;
DeviceMapping.Output00_02 := G_IO.O_StopPushButton;

END_PROGRAM

// ---- POUs/General/ErrorHandle.TcPOU
PROGRAM ErrorHandle
VAR
END_VAR

//===================================
//Machine Control
//===================================
G_MachineControl.bMainError := %MD1000 > 0;

//===================================
//Warning MD1005
//===================================

//===================================
//ST00 Conveyor
//===================================	

G_MachineControl.arrstStationControl[0].bError := %MD1008 > 0 OR %MD1009 > 0;

//===================================
//ST10 Barcode Scanner 
//===================================

G_MachineControl.arrstStationControl[1].bError := %MD1010 > 0;

//===================================
//ST20 Robot Pick & Place
//===================================

G_MachineControl.arrstStationControl[2].bError := %MD1020 > 0 OR %MD1021 > 0;

END_PROGRAM

// ---- POUs/Station/ST00_Conveyor/ST00_ChangeRecipe.TcPOU
PROGRAM ST00_ChangeRecipe
VAR
	iStep : INT;
END_VAR

END_PROGRAM

// ---- POUs/Station/ST00_Conveyor/ST00_Cylinder.TcPOU
PROGRAM ST00_Cylinder
VAR
	fbLifter: FB_DoubleActingCylinder;
	fbStopper: FB_DoubleActingCylinder;
END_VAR

IF NOT G_Manual.M_CheckIOUse THEN
	fbLifter(
		IN_bManualMode:= G_MachineControl.stMachineOperateMode.MANUAL, 
		IN_bAutoMode:= G_MachineControl.stMachineOperateMode.AUTO OR G_MachineControl.stMachineOperateMode.DRYRUN, 
		IN_bWork_IOTrig_Input:= G_Manual.M00_bLifterCylUp OR G_Home.H00_bLifterCylUp, 
		IN_bHome_IOTrig_Input:= G_Manual.M00_bLifterCylDown OR G_Home.H00_bLifterCylDown, 
		IN_bWork_PRGTrig:= G_Auto.A00_bLifterCylUp OR G_Home.H00_bLifterCylUp, 
		IN_bHome_PRGTrig:= G_Auto.A00_bLifterCylDown OR G_Home.H00_bLifterCylDown, 
		IN_bWork_Rs:= G_IO.I_LifterUp, 
		IN_bHome_Rs:= G_IO.I_LifterDown, 
		IN_tWork_Timeout:= T#2S, 
		IN_tHome_Timeout:= T#2S, 
		IN_tWork_DelayTime:= T#0S, 
		IN_tHome_DelayTime:= T#0S, 
		IN_bAlarmEnable:= TRUE, 
		IN_bReset:= G_MachineControl.bMachineReset, 
		IN_tWorkRsCheck:= T#300MS, 
		IN_tHomeRsCheck:= T#300MS, 
		OUT_bWork=> G_IO.O_LifterUp, 
		OUT_bHome=> G_IO.O_LifterDown, 
		OUT_bWorkDone=> G_Auto.A00_bLifterCylUpDone, 
		OUT_bWorkDone=> G_Home.H00_bLifterCylUpDone, 
		OUT_bWorkDone=> G_Manual.M00_bLifterCylUpDone, 
		OUT_bHomeDone=> G_Auto.A00_bLifterCylDownDone, 
		OUT_bHomeDone=> G_Home.H00_bLifterCylDownDone, 
		OUT_bHomeDone=> G_Manual.M00_bLifterCylDownDone, 
		OUT_bError=> , 
		OUT_sErrorStatus=> , 
		OUT_bWorkError=> G_Error.E00_LifterCylUp, 
		OUT_bHomeError=> G_error.E00_LifterCylDown, 
		OUT_bRSError=> , 
		OUT_bInputError=> );
		
	fbStopper(
		IN_bManualMode:= G_MachineControl.stMachineOperateMode.MANUAL, 
		IN_bAutoMode:= G_MachineControl.stMachineOperateMode.AUTO OR G_MachineControl.stMachineOperateMode.DRYRUN, 
		IN_bWork_IOTrig_Input:= G_Manual.M00_bStopperCylBlock OR G_Home.H00_bStopperCylBlock, 
		IN_bHome_IOTrig_Input:= G_Manual.M00_bStopperCylRelease OR G_Home.H00_bStopperCylRelease, 
		IN_bWork_PRGTrig:= G_Auto.A00_bStopperCylBlock OR G_Home.H00_bStopperCylBlock, 
		IN_bHome_PRGTrig:= G_Auto.A00_bStopperCylRelease OR G_Home.H00_bStopperCylRelease, 
		IN_bWork_Rs:= G_IO.I_LifterUp, 
		IN_bHome_Rs:= G_IO.I_LifterDown, 
		IN_tWork_Timeout:= T#2S, 
		IN_tHome_Timeout:= T#2S, 
		IN_tWork_DelayTime:= T#0S, 
		IN_tHome_DelayTime:= T#0S, 
		IN_bAlarmEnable:= TRUE, 
		IN_bReset:= G_MachineControl.bMachineReset, 
		IN_tWorkRsCheck:= T#300MS, 
		IN_tHomeRsCheck:= T#300MS, 
		OUT_bWork=> G_IO.O_LifterUp, 
		OUT_bHome=> G_IO.O_LifterDown, 
		OUT_bWorkDone=> G_Auto.A00_bStopperCylBlockDone, 
		OUT_bWorkDone=> G_Home.H00_bStopperCylBlockDone, 
		OUT_bWorkDone=> G_Manual.M00_bStopperCylBlockDone, 
		OUT_bHomeDone=> G_Auto.A00_bStopperCylReleaseDone, 
		OUT_bHomeDone=> G_Home.H00_bStopperCylReleaseDone, 
		OUT_bHomeDone=> G_Manual.M00_bStopperCylReleaseDone, 
		OUT_bError=> , 
		OUT_sErrorStatus=> , 
		OUT_bWorkError=> G_Error.E00_StopperCylBlock, 
		OUT_bHomeError=> G_error.E00_StopperCylRelease, 
		OUT_bRSError=> , 
		OUT_bInputError=> );
END_IF

END_PROGRAM

// ---- POUs/Station/ST00_Conveyor/ST00_Sequence.TcPOU
PROGRAM ST00_Sequence
VAR
END_VAR

END_PROGRAM

// ---- POUs/Station/ST10_BarcodeScanner/ST10_BarcodeScanner.TcPOU
PROGRAM ST10_BarcodeScanner
VAR
	fbCognexBarcodeScanner: FB_CognexBarcodeScanner;
END_VAR

fbCognexBarcodeScanner(
	In_bManualMode:= G_MachineControl.stMachineOperateMode.MANUAL,
	In_bAutoMode:= G_MachineControl.stMachineOperateMode.AUTO OR G_MachineControl.stMachineOperateMode.DRYRUN,
	In_timeScanTimer:= T#10S, 
	In_iResultByte:= 20, 
	In_ioDeviceFault := G_Scanner.In_Signal_Conveyor.In_GeneralFault,
	In_ioTriggerReady:= G_Scanner.In_Signal_Conveyor.In_TriggerReady, 
	In_ioTriggerAck:= G_Scanner.In_Signal_Conveyor.In_TriggerAck, 
	In_ioAcquiring:= G_Scanner.In_Signal_Conveyor.In_Acquiring, 
	In_ioArrayData:= G_Scanner.In_Signal_Conveyor.In_ResultData, 
	Out_bDeviceError=> G_Error.E10_BarcodeScannerDeviceError,
	Out_bErrScanTimeOut=> G_Error.E10_BarcodeTimeout, 
	Out_ioTriggerEnable=> G_Scanner.Out_Signal_Conveyor.Out_TriggerEnable, 
	Out_ioTrigger=> G_Scanner.Out_Signal_Conveyor.Out_Trigger, 
	Out_bEnableReady=> G_Manual.M10_bTriggerScannerEnableReady,
	Out_bEnableReady=> G_Auto.A10_bTriggerScannerEnableReady,
	Out_bTriggerDone=> G_Manual.M10_bTriggerScannerDone,
	Out_bTriggerDone=> G_Auto.A10_bTriggerScannerDone,
	Out_sAutoBarcode=> G_Auto.A10_sScannerBarcode, 
	Out_sManualBarcode=> G_Manual.M10_sScannerBarcode, 
	Out_GetBarcodeDone=> G_Auto.A10_bScannerResultDone,
	Out_GetBarcodeDone=> G_Manual.M10_bScannerResultDone, 
	InOut_bAutoTriggerEnable:= G_Auto.A10_bTriggerScannerEnable, 
	InOut_bManualTriggerEnable:= G_Manual.M10_bTriggerScannerEnable, 
	InOut_bAutoTrigger:= G_Auto.A10_bTriggerScanner,
	InOut_bManualTrigger:= G_Manual.M10_bTriggerScanner);

END_PROGRAM

// ---- POUs/Function Block/FB_CognexBarcodeScanner.TcPOU
FUNCTION_BLOCK FB_CognexBarcodeScanner
VAR_INPUT
	In_bManualMode		: BOOL; // Manual Mode
	In_bAutoMode		: BOOL; // Auto Mode
	In_timeScanTimer	: TIME;
	In_iResultByte		: INT;
	In_ioDeviceFault	: BOOL;
	In_ioTriggerReady	: BOOL;
	In_ioTriggerAck		: BOOL;
	In_ioAcquiring		: BOOL;
	In_ioArrayData		: ARRAY [1..480] OF BYTE;
END_VAR
VAR_OUTPUT
	Out_bDeviceError	: BOOL;
	Out_bErrScanTimeOut : BOOL;
	Out_ioTriggerEnable	: BOOL;
	Out_ioTrigger		: BOOL;
	Out_bEnableReady	: BOOL;
	Out_bTriggerDone	: BOOL;
	Out_sAutoBarcode	: STRING;
	Out_sManualBarcode	: STRING;
	Out_GetBarcodeDone	: BOOL;	
END_VAR
VAR_IN_OUT
	InOut_bAutoTriggerEnable	: BOOL;
	InOut_bManualTriggerEnable	: BOOL;
	InOut_bAutoTrigger			: BOOL;
	InOut_bManualTrigger		: BOOL;
END_VAR
VAR
	rTrig_TriggerEnable: R_TRIG;
	fTrig_TriggerEnable: F_TRIG;
	
	rTrig_Trigger: R_TRIG;
	iStepTriggerEnable	: INT;
	iStepTrigger 		: INT;
	iforCount			: INT;
	sChar				: STRING(1);
	tonTimeOut			: TON;
	sBarcode			: STRING;
END_VAR

// Device Error
Out_bDeviceError := In_ioDeviceFault;
rTrig_TriggerEnable(CLK:=(InOut_bAutoTriggerEnable AND In_bAutoMode) OR (InOut_bManualTriggerEnable AND In_bManualMode));
fTrig_TriggerEnable(CLK:=(InOut_bAutoTriggerEnable AND In_bAutoMode) OR (InOut_bManualTriggerEnable AND In_bManualMode));
	
rTrig_Trigger(CLK:=(InOut_bAutoTrigger AND In_bAutoMode) OR (InOut_bManualTrigger AND In_bManualMode));

Out_bEnableReady := In_ioTriggerReady;

// Enable Trigger
CASE iStepTriggerEnable OF
	
	0 :
		IF rTrig_TriggerEnable.Q THEN
			Out_ioTriggerEnable := TRUE;
			iStepTriggerEnable := 10;
		ELSIF fTrig_TriggerEnable.Q THEN
			Out_ioTriggerEnable := FALSE;
			Out_bTriggerDone := FALSE;
			iStepTriggerEnable := 100;
		END_IF
		
	10:
		IF In_ioTriggerReady THEN
			InOut_bAutoTriggerEnable := TRUE;
			iStepTriggerEnable := 0;
		ELSIF fTrig_TriggerEnable.Q THEN
			Out_ioTriggerEnable := FALSE;
			Out_bTriggerDone := FALSE;
			iStepTriggerEnable := 100;
		END_IF
		
	100:
		IF NOT In_ioTriggerReady THEN
			Out_bTriggerDone := FALSE;
			iStepTriggerEnable := 0;
		END_IF
		
END_CASE

CASE iStepTrigger OF
	
	0:
		IF rTrig_Trigger.Q THEN
			Out_bErrScanTimeOut := FALSE;
			IF In_ioTriggerReady THEN
				Out_bTriggerDone := FALSE;
				Out_GetBarcodeDone := FALSE;
				Out_ioTrigger := TRUE;
				iStepTrigger := 10;
			ELSE
				Out_bTriggerDone := FALSE;
				Out_GetBarcodeDone := FALSE;
				Out_ioTriggerEnable := FALSE;
				iStepTrigger := 100;
			END_IF
		END_IF
		
	10:
		IF In_ioTriggerAck AND In_ioAcquiring THEN
			sBarcode := '';
			IF In_bAutoMode THEN
				Out_sAutoBarcode := '';
			END_IF
			IF In_bManualMode THEN
				Out_sManualBarcode := '';
			END_IF
			iStepTrigger := 20;
		END_IF
	
	20: 
		tonTimeOut(IN:= TRUE, PT:= In_timeScanTimer);
		IF NOT In_ioAcquiring THEN
			tonTimeOut(IN:= FALSE);
			FOR iforCount:=1 TO In_iResultByte BY 1 DO
				IF In_ioArrayData[iforCount] <> 0 THEN
					sChar := F_ToCHR(STRING_TO_BYTE(CONCAT('16#',WORD_TO_HEXSTR(In_ioArrayData[iforCount], 1, FALSE))));
					sBarcode:= CONCAT(sBarcode,sChar);
					IF In_bAutoMode THEN
						Out_sAutoBarcode := sBarcode;
					END_IF
					IF In_bManualMode THEN
						Out_sManualBarcode := sBarcode;
					END_IF
				END_IF
			END_FOR
			iStepTrigger := 30;
		ELSIF tonTimeOut.Q THEN
			tonTimeOut(IN:= FALSE);
			IF In_bAutoMode THEN
				InOut_bAutoTrigger := FALSE;
			END_IF
			IF In_bManualMode THEN
				InOut_bManualTrigger := FALSE;
			END_IF
			Out_bTriggerDone := TRUE;
			Out_ioTrigger := FALSE;
			Out_bErrScanTimeOut := TRUE;
			iStepTrigger := 0;
		END_IF
		
	30:	
		Out_GetBarcodeDone := TRUE;
		Out_bTriggerDone := TRUE;
		IF In_bAutoMode THEN
			InOut_bAutoTrigger := FALSE;
		END_IF
		IF In_bManualMode THEN
			InOut_bManualTrigger := FALSE;
		END_IF
		Out_ioTrigger := FALSE;
		iStepTrigger := 0;
		
	100:
		IF In_bAutoMode THEN
			InOut_bAutoTriggerEnable := TRUE;
		END_IF
		IF In_bManualMode THEN
			InOut_bManualTriggerEnable := FALSE;
		END_IF
		iStepTrigger := 110;
	
	110:
		IF In_ioTriggerReady THEN
			Out_ioTrigger := TRUE;
			iStepTrigger := 10;
		END_IF	

END_CASE

END_FUNCTION_BLOCK

// ---- POUs/Station/ST10_BarcodeScanner/ST10_Sequence.TcPOU
PROGRAM ST10_Sequence
VAR
	arrStepStatus : ARRAY [1..100] OF STRING;
	arrStepUsedTime	: ARRAY [1..100] OF TIME;
	tonStepTimer : TON;
	iStep : INT;
	iMatching: INT;
	bStart: BOOL;
	Reset_RTrig: R_TRIG;
	sBarcode: STRING;
END_VAR

tonStepTimer();

bStart := (G_MachineControl.stMachineCurrentMode.AUTO_RUNNING OR
				G_MachineControl.stMachineCurrentMode.DRYRUN_RUNNING);
				
IF NOT G_MachineControl.arrstStationControl[1].bError THEN
	CASE iStep OF
			
		0://Ready
			IF bStart AND NOT G_MachineControl.arrstStationControl[1].bByPassStation
				AND NOT G_MachineControl.arrstStationControl[1].bJobDone THEN
				arrStepStatus[1] := 'Step 1: Trigger Read Barcode';
				tonStepTimer(IN:=TRUE, PT:=T#999999S);
				G_Auto.A10_sScannerBarcode := '';
				G_Auto.A10_bTriggerScanner := TRUE;
				iStep := 10;
			ELSIF bStart AND G_MachineControl.arrstStationControl[1].bByPassStation AND NOT G_MachineControl.arrstStationControl[1].bJobDone  THEN
				iStep := 999;
			END_IF
			
		10://Waiting scanner ack
			IF NOT G_Auto.A10_bScannerResultDone THEN
				iStep := 20;
			END_IF
			
		20://Waiting scanner result done
			IF G_Auto.A10_bScannerResultDone THEN
				G_Auto.A10_bTriggerScanner := FALSE;
				arrStepUsedTime[1] := tonStepTimer.ET;
				tonStepTimer(IN:=FALSE);
				sBarcode := G_Auto.A10_sScannerBarcode;
				iStep := 999;
			ELSIF G_Error.E10_BarcodeTimeout THEN
				G_Error.E10_BarcodeTimeout := FALSE;
				arrStepUsedTime[1] := tonStepTimer.ET;
				tonStepTimer(IN:=FALSE);
				arrStepStatus[2] := 'Step 2: Trigger Check at MES';
				arrStepUsedTime[2] := tonStepTimer.ET;
				iStep := 999;
			END_IF
			
		999://Job Done
			G_MachineControl.arrstStationControl[1].bJobDone := TRUE;
			iStep := 0;	
			
	END_CASE
	
ELSIF G_MachineControl.arrstStationControl[1].bError THEN
	
	//When error waiting reset
	Reset_RTrig(CLK := G_MachineControl.bMachineReset);
	IF Reset_RTrig.Q THEN
		G_Error.E10_BarcodeScannerDeviceError := FALSE;	
	    G_Error.E10_BarcodeTimeout := FALSE;					
	END_IF

END_IF

FOR iMatching := 1 TO 100 DO
	G_MachineControl.arrsST10StepStatus[iMatching] := arrStepStatus[iMatching];
	G_MachineControl.arrtimeST10StepTime[iMatching] := arrStepUsedTime[iMatching];
END_FOR

END_PROGRAM

// ---- POUs/Station/ST20_PickNPlace/Robot/ST20_RobotManualControl.TcPOU
PROGRAM ST20_RobotManualControl
VAR
	iRobotPowerOn	: INT;
	timeDone		: TIME;
	tonTimeOut		: TON;
	tondelay		: TON;
	robotProgramID : BYTE;
END_VAR

timeDone := T#70MS;

//============================	
//General
//============================
 
IF G_MachineControl.stMachineOperateMode.MANUAL THEN	
	IF G_Manual.M20_bRobotHome THEN
		G_Robot.RobotKukaStandard.bHome := TRUE;
		IF G_Robot.RobotKukaStandard.bHome THEN //Req Robot Home
			tondelay(IN:=TRUE,PT:=timeDone);
			IF G_Robot.RobotKukaStandard.bHomeDone AND tondelay.Q THEN
				tondelay(IN:=FALSE);
				G_Robot.RobotKukaStandard.bHome := FALSE;
				G_Manual.M20_bRobotHome	:= FALSE;
			END_IF
		END_IF
	END_IF
	IF G_Manual.M20_bRobotEnable THEN
		G_Robot.RobotKukaStandard.bEnable := TRUE;
		IF G_Robot.RobotKukaStandard.bEnable THEN //Req Robot Start
			tonTimeOut(IN:= TRUE, PT:= T#5S);
			IF G_Robot.RobotKukaStandard.bEnabled THEN
				tonTimeOut(IN:= FALSE);
			ELSIF tonTimeOut.Q THEN
				G_Error.E20_RobotFailServoOn := TRUE;
				tonTimeOut(IN:= FALSE);
			END_IF
		END_IF
	END_IF
 
	IF G_Manual.M20_bRobotStart THEN
		G_Robot.RobotKukaStandard.bStart := TRUE;
		IF G_Robot.RobotKukaStandard.bStart THEN //Req Robot Start
			IF G_Robot.RobotKukaStandard.bRunning THEN
				G_Robot.RobotKukaStandard.bStop := FALSE;
				//G_Manual.M20_bRobotStart := FALSE;
			END_IF
		END_IF
	END_IF
	IF G_Manual.M20_bRobotStop THEN
		G_Robot.RobotKukaStandard.bStop := TRUE;
		IF G_Robot.RobotKukaStandard.bStop THEN //Req Robot Stop
			G_Robot.RobotKukaStandard.bStart := FALSE;
			IF G_Robot.RobotKukaStandard.bStopped THEN
				G_Robot.RobotKukaStandard.bStop := FALSE;
				G_Manual.M20_bRobotStop := FALSE;
			END_IF			
		END_IF
	END_IF
	IF G_Manual.M20_bRobotReset THEN
		G_Robot.RobotKukaStandard.bReset := TRUE;
		IF G_Robot.RobotKukaStandard.bReset THEN //Req Robot Reset
			IF NOT G_Robot.RobotKukaStandard.bError THEN
				G_Robot.RobotKukaStandard.bReset := FALSE;
				G_Manual.M20_bRobotReset := FALSE;
			END_IF			
		END_IF
	END_IF
 
	IF G_Manual.M20_bRobotPause THEN
		G_Robot.RobotKukaStandard.bPause := TRUE;
		IF G_Robot.RobotKukaStandard.bPause THEN //Req Robot Pause
			IF G_Robot.RobotKukaStandard.bPaused THEN
				G_Robot.RobotKukaStandard.bPause := FALSE;
				G_Manual.M20_bRobotPause := FALSE;
			END_IF
		END_IF		
	END_IF
 
	IF G_Manual.M20_bRobotContinue THEN
		G_Robot.RobotKukaStandard.bContinue := TRUE;
		IF G_Robot.RobotKukaStandard.bContinue THEN //Req Robot Continue
			IF G_Robot.RobotKukaStandard.bRunning THEN
				G_Robot.RobotKukaStandard.bContinue := FALSE;
				G_Manual.M20_bRobotContinue := FALSE;
			END_IF
		END_IF
	END_IF

	IF G_Manual.M20_bRobotPowerOn THEN //Req Robot Power On (Enable, Start, Ready For Command
		CASE iRobotPowerOn OF
		0: //
			G_Robot.RobotKukaStandard.bStop	:= TRUE;
			tonDelay(IN:=TRUE, PT:=T#2S);
			IF tonDelay.Q THEN
				tonDelay(IN:=FALSE);
				iRobotPowerOn := 10;
			END_IF	
		10:
			G_Robot.RobotKukaStandard.bStop	:= FALSE;
			tonDelay(IN:=TRUE, PT:=T#2S);
			IF tonDelay.Q THEN
				tonDelay(IN:=FALSE);
				iRobotPowerOn := 20;
			END_IF
		20:
			G_Robot.RobotKukaStandard.bEnable	:= FALSE;
			IF NOT G_Robot.RobotKukaStandard.bEnable THEN
				iRobotPowerOn := 30;
			END_IF
		30:
			tonDelay(IN:=TRUE, PT:=T#2S);
			IF tonDelay.Q THEN
				tonDelay(IN:=FALSE);
				iRobotPowerOn := 40;
			END_IF
		40: //Servo On @ Enable
			G_Robot.RobotKukaStandard.bEnable	:= TRUE;
			G_Robot.RobotKukaStandard.bStop	:= FALSE; 
			iRobotPowerOn := 50;
		50:
			tonTimeOut(IN:= TRUE, PT:= T#5S);
			IF G_Robot.RobotKukaStandard.bEnabled THEN
				tonTimeOut(IN:= FALSE);
				iRobotPowerOn := 60;
			ELSIF tonTimeOut.Q THEN
				G_Error.E20_RobotFailServoOn := TRUE;
				tonTimeOut(IN:= FALSE);
				iRobotPowerOn := 40;
			END_IF
		60:
			G_Robot.RobotKukaStandard.bReset	:= TRUE;
			IF NOT G_Robot.RobotKukaStandard.bStopped THEN
				iRobotPowerOn := 70;
			END_IF
		70:
			G_Robot.RobotKukaStandard.bStart	:= FALSE;
			IF NOT G_Robot.RobotKukaStandard.bStart THEN
				iRobotPowerOn := 80;
			END_IF
		80: 
			G_Robot.RobotKukaStandard.bReset	:= FALSE;
			IF NOT G_Robot.RobotKukaStandard.bReset THEN
				iRobotPowerOn := 90;
			END_IF
		90: 	
			tonTimeOut(IN:=TRUE, PT:=T#1S);
			IF tonTimeOut.Q THEN
				tonTimeOut(IN:=FALSE);
				iRobotPowerOn := 100;
			END_IF
		100: //Robot start
			G_Robot.RobotKukaStandard.bStart := TRUE;
			iRobotPowerOn := 110;
		110: //Wait start
			tonTimeOut(IN:= TRUE, PT:= T#50S);
			IF G_Robot.RobotKukaStandard.bRunning THEN
				tonTimeOut(IN:=FALSE);
				iRobotPowerOn := 0;
				G_Manual.M20_bRobotPowerOn := FALSE;
			ELSIF tonTimeOut.Q THEN
				tonTimeOut(IN:=FALSE);
				G_Robot.RobotKukaStandard.bStart := FALSE;
				G_Error.E20_RobotFailStart := TRUE;	
				iRobotPowerOn := 100;
			END_IF
		END_CASE
	END_IF
	
	IF G_Manual.M20_bRobotStandbyPos THEN
		G_Robot.RobotKukaStandard.bStandbyPosition := TRUE;
		IF G_Robot.RobotKukaStandard.bStandbyPosition THEN //Robot Standby Position
			tondelay(IN:=TRUE,PT:=timeDone);
			IF G_Robot.RobotKukaStandard.bStandbyPositionDone AND tondelay.Q THEN
				tondelay(IN:=FALSE);
				G_Robot.RobotKukaStandard.bStandbyPosition := FALSE;
				G_Manual.M20_bRobotStandbyPos := FALSE;
			END_IF
		END_IF
	END_IF
 
	IF G_Manual.M20_bClearMessage THEN
		G_Robot.RobotKukaStandard.bClearMessage := TRUE;
		IF G_Robot.RobotKukaStandard.bClearMessage THEN //Robot Standby Position
			tondelay(IN:=TRUE,PT:=timeDone);
			IF G_Robot.RobotKukaStandard.bClearMessageDone AND tondelay.Q THEN
				tondelay(IN:=FALSE);
				G_Robot.RobotKukaStandard.bClearMessageDone := FALSE;
				G_Manual.M20_bClearMessage := FALSE;
			END_IF
		END_IF
	END_IF	
 
	IF G_Manual.M20_bRobotGripperOnOff AND NOT G_Robot.RobotKukaCmd.bRobotGripperOnDone THEN //Robot Gripper
		G_Robot.RobotKukaCmd.bRobotGripperOnOff := TRUE;
	ELSIF NOT G_Manual.M20_bRobotGripperOnOff AND G_Robot.RobotKukaCmd.bRobotGripperOnDone THEN
		G_Robot.RobotKukaCmd.bRobotGripperOnOff := FALSE;
	END_IF

	
//============================	
//Sequence
//============================
	//Robot Pallet Fiducial 1 
	IF G_Manual.M20_bRobotPalletFiducial1 THEN
		G_Robot.RobotKukaCmd.bRobotPalletFiducial1 := TRUE;
		IF G_Robot.RobotKukaCmd.bRobotPalletFiducial1 THEN
			tondelay(IN:=TRUE,PT:=timeDone);
			IF G_Robot.RobotKukaCmd.bRobotPalletFiducial1Done AND tondelay.Q THEN
				tondelay(IN:=FALSE);
				G_Robot.RobotKukaCmd.bRobotPalletFiducial1 := FALSE;
				G_Manual.M20_bRobotPalletFiducial1 := FALSE;
			END_IF
		END_IF
	END_IF

	//Robot Pallet Fiducial 2
	IF G_Manual.M20_bRobotPalletFiducial2 THEN
		G_Robot.RobotKukaCmd.rRobotPlace_X := G_Values.VA20_stPalletPosition.stFiducialDistance2Value.Xpos;
		G_Robot.RobotKukaCmd.rRobotPlace_Y := G_Values.VA20_stPalletPosition.stFiducialDistance2Value.Ypos;
		G_Robot.RobotKukaCmd.rRobotPlace_Z := 0; //G_Values.VA20_rTrayZaxisPick; 
		G_Robot.RobotKukaCmd.rRobotPlace_A := G_Values.VA20_stPalletPosition.stFiducialDistance2Value.Apos;
		G_Robot.RobotKukaCmd.bRobotPalletFiducial2 := TRUE;
		IF G_Robot.RobotKukaCmd.bRobotPalletFiducial2 THEN
			tondelay(IN:=TRUE,PT:=timeDone);
			IF G_Robot.RobotKukaCmd.bRobotPalletFiducial2Done AND tondelay.Q THEN
				tondelay(IN:=FALSE);
				G_Robot.RobotKukaCmd.bRobotPalletFiducial2 := FALSE;
				G_Manual.M20_bRobotPalletFiducial2 := FALSE;
			END_IF
		END_IF
	END_IF
	
	//Robot Tray Fiducial 1 
	IF G_Manual.M20_bRobotTrayFiducial1 THEN
		G_Robot.RobotKukaCmd.bRobotTrayFiducial1 := TRUE;
		IF G_Robot.RobotKukaCmd.bRobotTrayFiducial1 THEN
			tondelay(IN:=TRUE,PT:=timeDone);
			IF G_Robot.RobotKukaCmd.bRobotTrayFiducial1Done AND tondelay.Q THEN
				tondelay(IN:=FALSE);
				G_Robot.RobotKukaCmd.bRobotTrayFiducial1 := FALSE;
				G_Manual.M20_bRobotTrayFiducial1 := FALSE;
			END_IF
		END_IF
	END_IF
	
	//Robot Tray Fiducial 2
	IF G_Manual.M20_bRobotTrayFiducial2 THEN
		G_Robot.RobotKukaCmd.rRobotPlace_X := G_Values.VA20_stTrayPosition.stFiducialDistance2Value.Xpos;
		G_Robot.RobotKukaCmd.rRobotPlace_Y := G_Values.VA20_stTrayPosition.stFiducialDistance2Value.Ypos;
		G_Robot.RobotKukaCmd.rRobotPlace_Z := 0; 
		G_Robot.RobotKukaCmd.rRobotPlace_A := G_Values.VA20_stTrayPosition.stFiducialDistance2Value.Apos;
		G_Robot.RobotKukaCmd.bRobotTrayFiducial2 := TRUE;
		IF G_Robot.RobotKukaCmd.bRobotTrayFiducial2 THEN
			tondelay(IN:=TRUE,PT:=timeDone);
			IF G_Robot.RobotKukaCmd.bRobotTrayFiducial2Done AND tondelay.Q THEN
				tondelay(IN:=FALSE);
				G_Robot.RobotKukaCmd.bRobotTrayFiducial2 := FALSE;
				G_Manual.M20_bRobotTrayFiducial2 := FALSE;
			END_IF
		END_IF
	END_IF
	
	//Robot Pick PCBA
	IF G_Manual.M20_bRobotPickPCBAPos THEN
		IF G_Manual.M20_bWithVisionData AND G_Vision.V20_stResultTrayPosition.Xpos > 0 AND G_Vision.V20_stResultTrayPosition.Ypos > 0 THEN 
			G_Robot.RobotKukaCmd.rRobotPlace_X := G_Vision.V20_stResultTrayPosition.Xpos;
			G_Robot.RobotKukaCmd.rRobotPlace_Y := G_Vision.V20_stResultTrayPosition.Ypos;
			G_Robot.RobotKukaCmd.rRobotPlace_Z := G_Values.VA20_rTrayZaxisPick; 
			G_Robot.RobotKukaCmd.rRobotPlace_A := G_Vision.V20_stResultTrayPosition.Apos;
		ELSE 
			G_Robot.RobotKukaCmd.rRobotPlace_X := G_Values.VA20_stTrayPosition.stPocket.Xpos;
			G_Robot.RobotKukaCmd.rRobotPlace_Y := G_Values.VA20_stTrayPosition.stPocket.Ypos;
			G_Robot.RobotKukaCmd.rRobotPlace_Z := G_Values.VA20_rTrayZaxisPick; 
			G_Robot.RobotKukaCmd.rRobotPlace_A := G_Values.VA20_stTrayPosition.stPocket.Apos;
		END_IF
		G_Robot.RobotKukaCmd.bRobotPickPCBA := TRUE;
		IF G_Robot.RobotKukaCmd.bRobotPickPCBA THEN //Robot Pick PCBA 
			tondelay(IN:=TRUE,PT:=timeDone);
			IF G_Robot.RobotKukaCmd.bRobotPickPCBADone AND tondelay.Q THEN
				tondelay(IN:=FALSE);
				G_Robot.RobotKukaCmd.bRobotPickPCBA := FALSE;
				G_Manual.M20_bRobotPickPCBAPos := FALSE;
			END_IF
		END_IF
	END_IF
	
	//Robot Place PCBA
	IF G_Manual.M20_bRobotPlacePCBAPos THEN
		IF G_Manual.M20_bWithVisionData AND G_Vision.V20_stResultPalletPosition.Xpos > 0 AND G_Vision.V20_stResultPalletPosition.Ypos > 0 THEN 
			G_Robot.RobotKukaCmd.rRobotPlace_X := G_Vision.V20_stResultPalletPosition.Xpos;
			G_Robot.RobotKukaCmd.rRobotPlace_Y := G_Vision.V20_stResultPalletPosition.Ypos;
			G_Robot.RobotKukaCmd.rRobotPlace_Z := G_Values.VA20_rPalletZaxisPlace; 
			G_Robot.RobotKukaCmd.rRobotPlace_A := G_Vision.V20_stResultPalletPosition.Apos;
		ELSE 
			G_Robot.RobotKukaCmd.rRobotPlace_X := G_Values.VA20_stPalletPosition.stPocket.Xpos;
			G_Robot.RobotKukaCmd.rRobotPlace_Y := G_Values.VA20_stPalletPosition.stPocket.Ypos;
			G_Robot.RobotKukaCmd.rRobotPlace_Z := G_Values.VA20_rPalletZaxisPlace; 
			G_Robot.RobotKukaCmd.rRobotPlace_A := G_Values.VA20_stPalletPosition.stPocket.Apos;
		END_IF
		G_Robot.RobotKukaCmd.bRobotPlacePCBA := TRUE;
		IF G_Robot.RobotKukaCmd.bRobotPlacePCBA THEN //Robot Place PCBA 
			tondelay(IN:=TRUE,PT:=timeDone);
			IF G_Robot.RobotKukaCmd.bRobotPlacePCBADone AND tondelay.Q THEN
				tondelay(IN:=FALSE);
				G_Robot.RobotKukaCmd.bRobotPlacePCBA := FALSE;
				G_Manual.M20_bRobotPlacePCBAPos := FALSE;
			END_IF
		END_IF
	END_IF
	
	//Robot Standby At Pallet
	IF G_Manual.M20_bRobotAtStandbyPallet THEN
		G_Robot.RobotKukaCmd.bRobotStandbyAtPallet := TRUE;
		IF G_Robot.RobotKukaCmd.bRobotStandbyAtPallet THEN
			tondelay(IN:=TRUE,PT:=timeDone);
			IF G_Robot.RobotKukaCmd.bRobotStandbyAtPalletDone AND tondelay.Q THEN
				tondelay(IN:=FALSE);
				G_Robot.RobotKukaCmd.bRobotStandbyAtPallet := FALSE;
				G_Manual.M20_bRobotAtStandbyPallet := FALSE;
			END_IF
		END_IF
	END_IF
	
	//Robot Standby At Tray
	IF G_Manual.M20_bRobotAtStandbyTray THEN
		G_Robot.RobotKukaCmd.bRobotStandbyAtTray := TRUE;
		IF G_Robot.RobotKukaCmd.bRobotStandbyAtTray THEN
			tondelay(IN:=TRUE,PT:=timeDone);
			IF G_Robot.RobotKukaCmd.bRobotStandbyAtTrayDone AND tondelay.Q THEN
				tondelay(IN:=FALSE);
				G_Robot.RobotKukaCmd.bRobotStandbyAtTray := FALSE;
				G_Manual.M20_bRobotAtStandbyTray := FALSE;
			END_IF
		END_IF
	END_IF
	
 
	IF G_Manual.M20_bChangeRobotProgramID THEN
		G_Robot.RobotKukaStandard.bAppID0 := BIT_TO_BOOL(G_Manual.M20_byteRobotProgramID.0);
		G_Robot.RobotKukaStandard.bAppID1 := BIT_TO_BOOL(G_Manual.M20_byteRobotProgramID.1);
		G_Robot.RobotKukaStandard.bAppID2 := BIT_TO_BOOL(G_Manual.M20_byteRobotProgramID.2);
		G_Manual.M20_bChangeRobotProgramID := FALSE;
	END_IF
END_IF

END_PROGRAM

// ---- POUs/Station/ST20_PickNPlace/Robot/ST20_RobotSequence.TcPOU
PROGRAM ST20_RobotSequence
VAR
	bEStopTriggered			: BOOL;
	iStepActiveRobot		: INT;
	iStepInitialize			: INT;
	iStepChangeRobotProgram : INT;
	tonTimeOut				: TON;
	tonDelay				: TON;
	Reset_RTRIG				: R_TRIG;
	iStepCheckDatum			: INT;
END_VAR

//timeTimeOut := T#20S;

//===================================
//Robot Initialize
//===================================

IF NOT G_MachineControl.arrstStationControl[2].bError THEN

	CASE iStepInitialize OF
		
		 0:
		 	IF G_Auto.A20_bRobotInitialize AND NOT G_MachineControl.stMachineCurrentMode.MANUAL_RUNNING THEN
				G_Auto.A20_bRobotInitializeDone  := FALSE;
				iStepInitialize := 10;
			END_IF
			
		10: //Robot Stop
			G_Robot.RobotKukaStandard.bStop := TRUE;
			G_Robot.RobotKukaCmd.bRobotTrayFiducial1 := FALSE;
			G_Robot.RobotKukaCmd.bRobotTrayFiducial2 := FALSE;
			G_Robot.RobotKukaCmd.bRobotPalletFiducial1 := FALSE;
			G_Robot.RobotKukaCmd.bRobotPalletFiducial2 := FALSE;
			G_Robot.RobotKukaCmd.bRobotPickPCBA := FALSE;
			G_Robot.RobotKukaCmd.bRobotPlacePCBA := FALSE;
			G_Robot.RobotKukaCmd.bRobotStandbyAtPallet := FALSE;
			G_Robot.RobotKukaCmd.bRobotStandbyAtTray := FALSE;
			G_Robot.RobotKukaStandard.bHome := FALSE;
			G_Robot.RobotKukaStandard.bStandbyPosition := FALSE;
			tonDelay(IN:=TRUE, PT:=T#2S);
			IF tonDelay.Q THEN
				tonDelay(IN:=FALSE);
				iStepInitialize := 20;
			END_IF	
			
		20:
			G_Robot.RobotKukaStandard.bStop	:= FALSE;
			tonDelay(IN:=TRUE, PT:=T#2S);
			IF tonDelay.Q THEN
				tonDelay(IN:=FALSE);
				iStepInitialize := 30;
			END_IF
			
		30:
			G_Robot.RobotKukaStandard.bEnable	:= FALSE;
			IF NOT G_Robot.RobotKukaStandard.bEnable THEN
				iStepInitialize := 40;
			END_IF
			
		40:
			tonDelay(IN:=TRUE, PT:=T#2S);
			IF tonDelay.Q THEN
				tonDelay(IN:=FALSE);
				iStepInitialize := 50;
			END_IF
			
		50: //Servo On @ Enable
			G_Robot.RobotKukaStandard.bEnable	:= TRUE;
			G_Robot.RobotKukaStandard.bStop	:= FALSE; 
			iStepInitialize := 60;
			
		60:
			tonTimeOut(IN:= TRUE, PT:= T#5S);
			IF G_Robot.RobotKukaStandard.bEnabled THEN
				tonTimeOut(IN:= FALSE);
				iStepInitialize := 70;
			ELSIF tonTimeOut.Q THEN
				G_Error.E20_RobotFailServoOn := TRUE;
				tonTimeOut(IN:= FALSE);
				iStepInitialize := 50;
			END_IF
			
		70:
			G_Robot.RobotKukaStandard.bReset	:= TRUE;
			IF NOT G_Robot.RobotKukaStandard.bStopped THEN
 				iStepInitialize := 80;
			END_IF
			
		80:
			G_Robot.RobotKukaStandard.bStart	:= FALSE;
			IF NOT G_Robot.RobotKukaStandard.bStart THEN
 				iStepInitialize := 90;
			END_IF
			
		90: 
			G_Robot.RobotKukaStandard.bReset	:= FALSE;
			IF NOT G_Robot.RobotKukaStandard.bReset THEN
 				iStepInitialize := 100;
			END_IF
			
		100: //Robot program
			G_Robot.RobotKukaStandard.bAppID0 := TRUE;
			G_Robot.RobotKukaStandard.bAppID1 := FALSE;
			G_Robot.RobotKukaStandard.bAppID2 := FALSE;
			iStepChangeRobotProgram := 110;
			
		110: 	
			tonTimeOut(IN:=TRUE, PT:=T#1S);
			IF tonTimeOut.Q THEN
				tonTimeOut(IN:=FALSE);
				iStepInitialize := 120;
			END_IF
			
		120: //Robot start
			G_Robot.RobotKukaStandard.bStart := TRUE;
			iStepInitialize := 130;
					
		130: //Wait start
			tonTimeOut(IN:= TRUE, PT:= T#50S);
			IF G_Robot.RobotKukaStandard.bRunning THEN
				tonTimeOut(IN:=FALSE);
				iStepInitialize := 140;
			ELSIF tonTimeOut.Q THEN
				tonTimeOut(IN:=FALSE);
				G_Robot.RobotKukaStandard.bStart := FALSE;
				G_Error.E20_RobotFailStart := TRUE;
				G_Error.E20_RobotFailToInitialize := TRUE;	
				iStepInitialize := 120;
			END_IF
			
		140: //Robot Home
			G_Robot.RobotKukaStandard.bHome := TRUE;
			iStepInitialize := 150;
			
		150:
			IF NOT G_Robot.RobotKukaStandard.bHomeDone THEN
				iStepInitialize := 160;
			END_IF

		160: //Wait home
			tonTimeOut(IN:= TRUE, PT:= T#500S);
			IF G_Robot.RobotKukaStandard.bHomeDone THEN
				G_Robot.RobotKukaStandard.bHome := FALSE;
				tonTimeOut(IN:=FALSE);
				iStepInitialize := 999;	
			ELSIF tonTimeOut.Q THEN
				tonTimeOut(IN:=FALSE);
				G_Robot.RobotKukaStandard.bHome := FALSE;
				G_Error.E20_RobotFailHome := TRUE;
				G_Error.E20_RobotFailToInitialize := TRUE;	
				iStepInitialize := 140;
			END_IF				
		
		999: 
			G_Auto.A20_bRobotInitialize := FALSE;
			G_Auto.A20_bRobotInitializeDone  := TRUE;
			iStepInitialize := 0;			
	END_CASE

ELSE
	
	Reset_RTRIG(CLK := G_MachineControl.bMachineReset);
	IF Reset_RTRIG.Q THEN
		G_Error.E20_RobotFailHome 			:= FALSE;
		G_Error.E20_RobotFailStart			:= FALSE;
		G_Error.E20_RobotFailServoOn		:= FALSE;
		G_Error.E20_RobotFailToInitialize 	:= FALSE;
	END_IF
	
END_IF

//===================================
//Robot Recovery
//===================================

IF G_Error.E_EmgStop OR G_Robot.RobotKukaStandard.bEstopON THEN
	bEStopTriggered := TRUE;
END_IF

Reset_RTrig(CLK := G_MachineControl.bMachineReset);
IF Reset_RTrig.Q AND G_Robot.RobotKukaStandard.bAcknowledged THEN
	iStepActiveRobot := 10;
	bEStopTriggered := FALSE;
	G_Error.E20_RobotFailHome 			:= FALSE;
	G_Error.E20_RobotFailStart			:= FALSE;
	G_Error.E20_RobotFailServoOn		:= FALSE;
	G_Error.E20_RobotFailToInitialize 	:= FALSE;
END_IF

CASE iStepActiveRobot OF	
			
		10:
			G_Robot.RobotKukaStandard.bEnable	:= FALSE;
			G_Robot.RobotKukaStandard.bContinue	:= FALSE;
			G_Robot.RobotKukaStandard.bStart	:= FALSE;
			IF NOT G_Robot.RobotKukaStandard.bEnable THEN
				iStepActiveRobot := 20;
			END_IF
			
		20:
			tonDelay(IN:=TRUE, PT:=T#2S);
			IF tonDelay.Q THEN
				tonDelay(IN:=FALSE);
				iStepActiveRobot := 30;
			END_IF
			
		30: //Servo On @ Enable
			G_Robot.RobotKukaStandard.bEnable	:= TRUE;
			G_Robot.RobotKukaStandard.bStop	:= FALSE; 
			iStepActiveRobot := 40;
			
		40:
			tonTimeOut(IN:= TRUE, PT:= T#5S);
			IF G_Robot.RobotKukaStandard.bEnabled THEN
				tonTimeOut(IN:= FALSE);
				iStepActiveRobot := 50;
			ELSIF tonTimeOut.Q THEN
				G_Error.E20_RobotFailServoOn := TRUE;
				tonTimeOut(IN:= FALSE);
				iStepActiveRobot := 30;
			END_IF
			
		50:
		 	IF G_Robot.RobotKukaStandard.bPaused THEN
				G_Robot.RobotKukaStandard.bContinue	:= TRUE;
				IF G_Robot.RobotKukaStandard.bRunning THEN
					iStepActiveRobot := 60;
				END_IF
			END_IF
			
			IF NOT G_Robot.RobotKukaStandard.bPaused THEN
				G_Robot.RobotKukaStandard.bStart	:= TRUE;
				IF G_Robot.RobotKukaStandard.bRunning THEN
					iStepActiveRobot := 60;
				END_IF
			END_IF

			
		60:
			G_Robot.RobotKukaStandard.bContinue	:= FALSE;
			IF NOT G_Robot.RobotKukaStandard.bContinue THEN
 				iStepActiveRobot := 0;
			END_IF
				
END_CASE

//===================================
//Robot Check Datum
//===================================
 
IF NOT G_MachineControl.arrstStationControl[2].bError THEN
	CASE iStepCheckDatum OF
			 0:
				IF G_Auto.A20_bRobotCheckDatum AND NOT G_MachineControl.stMachineCurrentMode.MANUAL_RUNNING THEN //need to add signal with workspace R1 working or not 
					G_Auto.A20_bRobotCheckDatumDone := FALSE;
					iStepCheckDatum := 10;
				END_IF
			10: //Robot Datum Position
				G_Robot.RobotKukaCmd.bRobotCheckDatum := TRUE;
				iStepCheckDatum := 20;
			20:
				IF NOT G_Robot.RobotKukaCmd.bRobotCheckDatumDone THEN
					iStepCheckDatum := 30;
				END_IF
			30: //Wait datum position
				tonTimeOut(IN:= TRUE, PT:= T#500S);
				IF G_Robot.RobotKukaCmd.bRobotCheckDatumDone THEN
					G_Robot.RobotKukaCmd.bRobotCheckDatum := FALSE;
					tonTimeOut(IN:=FALSE);
					iStepCheckDatum := 40;	
				ELSIF tonTimeOut.Q THEN
					tonTimeOut(IN:=FALSE);
					G_Robot.RobotKukaCmd.bRobotCheckDatum := FALSE;
					G_Error.E20_RobotFailDatumPos := TRUE;	
					iStepCheckDatum := 10;
				END_IF
 
			40: //Vision capture datum
				G_Vision.V20_bRespone := FALSE;
				G_Vision.V20_sSendCmd := 'TRG,0'; //may change based on vision team
				G_Vision.V20_bTrigger := TRUE;				
				iStepCheckDatum := 50;
			50: //Waiting vision capture done
				tonTimeOut(IN:= TRUE,PT:= T#90S);
				IF G_Vision.V20_bRespone THEN
					G_Vision.V20_bTrigger := FALSE;
					tonTimeOut(IN:= FALSE);
					iStepCheckDatum := 60;
				ELSIF tonTimeOut.Q THEN
					tonTimeOut(IN:= FALSE);
					G_Error.E20_VisionTimeOutDatumCheck := TRUE;
					iStepCheckDatum := 40;
				END_IF	
			//60: // Result of vision - Pop out  succefully or not
			60:
				G_Values.VA20_sDatumVisionResultStatus := G_Vision.V20_sDatumVisionResultStatus;
				G_Values.VA20_stDatumVisionResultPos := G_Vision.V20_stDatumVisionResultPos;					
				iStepCheckDatum := 999;
			999: 
				G_Auto.A20_bRobotCheckDatum := FALSE;
				G_Auto.A20_bRobotCheckDatumDone  := TRUE;
				iStepCheckDatum := 0;			
		END_CASE
 
ELSE
	Reset_RTRIG(CLK := G_MachineControl.bMachineReset);
	IF Reset_RTRIG.Q THEN
		G_Error.E40_RobotFailDatumPos 		:= FALSE;
		G_Error.E40_VisionTimeOutDatumCheck	:= FALSE;
	END_IF
END_IF

END_PROGRAM

// ---- POUs/Station/ST20_PickNPlace/TrayLoader/ST20_BarcodeScanner.TcPOU
PROGRAM ST20_BarcodeScanner
VAR
	fbCognexBarcodeScanner: FB_CognexBarcodeScanner;
END_VAR

fbCognexBarcodeScanner(
	In_bManualMode:= G_MachineControl.stMachineOperateMode.MANUAL,
	In_bAutoMode:= G_MachineControl.stMachineOperateMode.AUTO OR G_MachineControl.stMachineOperateMode.DRYRUN,
	In_timeScanTimer:= T#10S, 
	In_iResultByte:= 20, 
	In_ioDeviceFault := G_Scanner.In_Signal_Tray.In_GeneralFault,
	In_ioTriggerReady:= G_Scanner.In_Signal_Tray.In_TriggerReady, 
	In_ioTriggerAck:= G_Scanner.In_Signal_Tray.In_TriggerAck, 
	In_ioAcquiring:= G_Scanner.In_Signal_Tray.In_Acquiring, 
	In_ioArrayData:= G_Scanner.In_Signal_Tray.In_ResultData, 
	Out_bDeviceError=> G_Error.E20_BarcodeScannerDeviceError,
	Out_bErrScanTimeOut=> G_Error.E20_BarcodeTimeout, 
	Out_ioTriggerEnable=> G_Scanner.Out_Signal_Tray.Out_TriggerEnable, 
	Out_ioTrigger=> G_Scanner.Out_Signal_Tray.Out_Trigger, 
	Out_bEnableReady=> G_Manual.M20_bTriggerScannerEnableReady,
	Out_bEnableReady=> G_Auto.A20_bTriggerScannerEnableReady,
	Out_bTriggerDone=> G_Manual.M20_bTriggerScannerDone,
	Out_bTriggerDone=> G_Auto.A20_bTriggerScannerDone,
	Out_sAutoBarcode=> G_Auto.A20_sScannerBarcode, 
	Out_sManualBarcode=> G_Manual.M20_sScannerBarcode, 
	Out_GetBarcodeDone=> G_Auto.A20_bScannerResultDone,
	Out_GetBarcodeDone=> G_Manual.M20_bScannerResultDone, 
	InOut_bAutoTriggerEnable:= G_Auto.A20_bTriggerScannerEnable, 
	InOut_bManualTriggerEnable:= G_Manual.M20_bTriggerScannerEnable, 
	InOut_bAutoTrigger:= G_Auto.A20_bTriggerScanner,
	InOut_bManualTrigger:= G_Manual.M20_bTriggerScanner);

END_PROGRAM

// ---- POUs/Station/ST20_PickNPlace/TrayLoader/ST20_TraySequence.TcPOU
PROGRAM ST20_TraySequence
VAR
	arrStepStatus : ARRAY [1..100] OF STRING;
	arrStepUsedTime	: ARRAY [1..100] OF TIME;
	tonStepTimer : TON;
	iStep : INT;
	iMatching: INT;
	bStart: BOOL;
	sBarcode: STRING;
END_VAR

tonStepTimer();

bStart := (G_MachineControl.stMachineCurrentMode.AUTO_RUNNING OR
				G_MachineControl.stMachineCurrentMode.DRYRUN_RUNNING);

//New Tray Procesee
CASE iStep OF
		
	0://Ready
		IF bStart AND G_Auto.A20_bIsNewTray THEN
			G_Auto.A20_bTriggerScanner := TRUE;
			iStep := 10;
		END_IF
		
	10://Waiting scanner ack
		IF NOT G_Auto.A20_bScannerResultDone THEN
			iStep := 20;
		END_IF
		
	20://Waiting scanner result done
		IF G_Auto.A20_bScannerResultDone THEN
			sBarcode := G_Auto.A20_sScannerBarcode;
			iStep := 30;
		ELSIF G_Error.E20_BarcodeTimeout THEN
			G_Error.E20_BarcodeTimeout := FALSE;
			G_Auto.A20_bTrayReady := FALSE;
			G_Auto.A20_bMESPass := FALSE;
			G_Auto.A20_bMESCheckDone := TRUE;
			iStep := 40;
		END_IF
		
	30://Trigger check at MES
		arrStepStatus[2] := 'Step 2: Trigger Check at MES';
		G_Auto.A20_bMESPass := FALSE;
		G_Auto.A20_bMESCheckDone := FALSE;
		G_Auto.A20_bMESCheck := TRUE;
		iStep := 40;	
		
	40://Waiting check at MES done
		IF G_Auto.A20_bMESCheckDone THEN
			G_Auto.A20_bMESCheck := FALSE;
			IF G_Auto.A20_bMESPass THEN
				G_Auto.A20_bTrayReady := TRUE;
				G_Auto.A20_bIsNewTray := FALSE;
				iStep := 999;	
			ELSE
				G_Auto.A20_bTrayReady := FALSE;	
				G_Auto.A20_bTrayFinish := TRUE;
				iStep := 0;	
			END_IF
		END_IF
		
	999://Job Done
		iStep := 0;	
		
END_CASE

END_PROGRAM

// ---- POUs/Station/ST20_PickNPlace/ST20_ChangeRecipe.TcPOU
PROGRAM ST20_ChangeRecipe
VAR
	tonTimeOut		: TON;
	tonDelay		: TON;
	Reset_RTRIG		: R_TRIG;
	iStepChangeRobotProgram : INT;
END_VAR

//===================================
//Robot Change Program
//===================================
IF NOT G_MachineControl.arrstStationControl[2].bError THEN
 
	CASE iStepChangeRobotProgram OF
		 0:
		 	IF G_Auto.A20_bRobotChangeRecipe AND NOT G_MachineControl.stMachineCurrentMode.MANUAL_RUNNING THEN
				G_Auto.A20_bRobotChangeRecipeDone  := FALSE;
				iStepChangeRobotProgram := 10;
			END_IF
		10: //
			G_Robot.RobotKukaStandard.bStop	:= TRUE;
			tonDelay(IN:=TRUE, PT:=T#2S);
			IF tonDelay.Q THEN
				tonDelay(IN:=FALSE);
				iStepChangeRobotProgram := 20;
			END_IF	
		20:
			G_Robot.RobotKukaStandard.bStop	:= FALSE;
			tonDelay(IN:=TRUE, PT:=T#2S);
			IF tonDelay.Q THEN
				tonDelay(IN:=FALSE);
				iStepChangeRobotProgram := 30;
			END_IF
		30:
			G_Robot.RobotKukaStandard.bReset	:= TRUE;
			IF NOT G_Robot.RobotKukaStandard.bStopped THEN
				iStepChangeRobotProgram := 40;
			END_IF
		40:
			G_Robot.RobotKukaStandard.bStart	:= FALSE;
			IF NOT G_Robot.RobotKukaStandard.bStart THEN
				iStepChangeRobotProgram := 50;
			END_IF
		50: 
			G_Robot.RobotKukaStandard.bReset	:= FALSE;
			IF NOT G_Robot.RobotKukaStandard.bReset THEN
				iStepChangeRobotProgram := 60;
			END_IF	
		60: //Robot program
			G_Robot.RobotKukaStandard.bAppID0 := BIT_TO_BOOL(G_Values.VA20_byteRobotProgramID.0);
			G_Robot.RobotKukaStandard.bAppID1 := BIT_TO_BOOL(G_Values.VA20_byteRobotProgramID.1);
			G_Robot.RobotKukaStandard.bAppID2 := BIT_TO_BOOL(G_Values.VA20_byteRobotProgramID.2);
			iStepChangeRobotProgram := 70;
		70: 	
			tonTimeOut(IN:=TRUE, PT:=T#1S);
			IF tonTimeOut.Q THEN
				tonTimeOut(IN:=FALSE);
				iStepChangeRobotProgram := 80;
			END_IF
		80: //Robot start
			G_Robot.RobotKukaStandard.bStart := TRUE;
			iStepChangeRobotProgram := 90;
		90: //Wait start
			tonTimeOut(IN:= TRUE, PT:= T#50S);
			IF G_Robot.RobotKukaStandard.bRunning THEN
				tonTimeOut(IN:=FALSE);
				iStepChangeRobotProgram := 999;
			ELSIF tonTimeOut.Q THEN
				tonTimeOut(IN:=FALSE);
				G_Robot.RobotKukaStandard.bStart := FALSE;
				G_Error.E20_RobotFailStart := TRUE;
				iStepChangeRobotProgram := 80;
			END_IF	
		999: 
			G_Auto.A20_bRobotChangeRecipe := FALSE;
			G_Auto.A20_bRobotChangeRecipeDone  := TRUE;
			iStepChangeRobotProgram := 0;			
	END_CASE
 
ELSE
	Reset_RTRIG(CLK := G_MachineControl.bMachineReset);
	IF Reset_RTRIG.Q THEN
		G_Error.E20_RobotFailHome 			:= FALSE;
		G_Error.E20_RobotFailStart			:= FALSE;
		G_Error.E20_RobotFailServoOn		:= FALSE;
		G_Error.E20_RobotFailToInitialize 	:= FALSE;
	END_IF
END_IF

END_PROGRAM

// ---- POUs/Station/ST20_PickNPlace/ST20_Home.TcPOU
PROGRAM ST20_Home
VAR
	bStart		: BOOL;
	iStepHome	: INT;
	tonTimeOut	: TON;
	Reset_RTRIG	: R_TRIG;
END_VAR

//===================================
//Home Sequence
//===================================
bStart := ((G_MachineControl.stMachineCurrentMode.INITIALIZE) OR
			 (G_MachineControl.stMachineCurrentMode.AUTO_RUNNING) OR
			 (G_MachineControl.stMachineCurrentMode.MANUAL_RUNNING));
			 
IF NOT G_MachineControl.arrstStationControl[2].bError  THEN
	
	CASE iStepHome OF
		0://Checking condition
			IF bStart AND NOT G_MachineControl.arrstStationControl[2].bByPassStation AND G_Home.H20_bHome THEN //need to add robot interlock for another robot
				G_Home.H20_bHomeDone := FALSE;
				iStepHome := 10;
			ELSIF bStart AND G_MachineControl.arrstStationControl[2].bByPassStation AND G_Home.H20_bHome THEN //need to add robot interlock for another robot
				G_Home.H20_bHome	:= FALSE;
				G_Home.H20_bHomeDone := TRUE;
				iStepHome := 0;
			END_IF
		
		10:
			G_Auto.A20_bRobotInitializeDone  := FALSE;
			G_Auto.A20_bRobotInitialize := TRUE;
			iStepHome := 20;
			
		20:
			IF G_Auto.A20_bRobotInitializeDone THEN
				iStepHome := 999;
			END_IF
		
		999: //Home Done
			G_Home.H20_bHome := FALSE;
			G_Home.H20_bHomeDone  := TRUE;
			iStepHome := 0;	
			
	END_CASE

ELSIF G_MachineControl.arrstStationControl[2].bError THEN
	Reset_RTrig(CLK := G_MachineControl.bMachineReset);
	IF Reset_RTrig.Q THEN
		G_Error.E20_RobotFailHome 			:= FALSE;
		G_Error.E20_RobotFailStart			:= FALSE;
		G_Error.E20_RobotFailServoOn		:= FALSE;
		G_Error.E20_RobotFailToInitialize	:= FALSE;
	END_IF
	
END_IF

END_PROGRAM

// ---- POUs/Station/ST20_PickNPlace/ST20_Sequence.TcPOU
PROGRAM ST20_Sequence
VAR
	arrStepStatus : ARRAY [1..100] OF STRING;
	arrStepUsedTime	: ARRAY [1..100] OF TIME;
	tonStepTimer : TON;
	iStep : int;
	bStart: BOOL;
	iMatching: INT;
	tonTimeOut : TON;
	tonDelay : TON;
	tTimeOut : TIME;
END_VAR

tonStepTimer();

bStart := (G_MachineControl.stMachineCurrentMode.AUTO_RUNNING OR
			G_MachineControl.stMachineCurrentMode.DRYRUN_RUNNING);

IF NOT G_MachineControl.arrstStationControl[2].bError THEN
				
	CASE iStep OF
		
		0: //Ready
			IF bStart AND NOT G_MachineControl.arrstStationControl[2].bByPassStation AND G_Auto.A20_bPalletReady AND G_Auto.A10_sScannerBarcode <> '' AND NOT G_MachineControl.arrstStationControl[2].bJobDone THEN
				G_Auto.A20_bRobotAtStandbyPallet := FALSE;
				iStep := 10;
			ELSIF bStart AND NOT G_MachineControl.arrstStationControl[2].bByPassStation AND NOT G_Auto.A20_bPalletReady AND NOT G_Auto.A20_bRobotAtStandbyPallet THEN
				iStep := 1000; //go to standby at pallet
			ELSIF bStart AND G_MachineControl.arrstStationControl[2].bByPassStation OR (G_Auto.A20_bPalletReady AND G_Auto.A10_sScannerBarcode <> '') AND NOT G_MachineControl.arrstStationControl[2].bJobDone THEN
				iStep := 999;
			END_IF
			
		10: //Robot move to pallet fiducial 1
			arrStepStatus[1] := 'Step 1: Robot go to pallet fiducial 1';
			tonStepTimer(IN:=TRUE, PT:=T#999999S);
			G_Robot.RobotKukaCmd.bRobotPalletFiducial1 := TRUE;
			iStep := 20; 
			
		20:
			IF NOT G_Robot.RobotKukaCmd.bRobotPalletFiducial1Done THEN
				iStep := 30;
			END_IF
			
		30://Robot move pallet fiducial 1 done
			tonTimeOut(IN:= TRUE,PT:= tTimeOut);
			IF G_Robot.RobotKukaCmd.bRobotPalletFiducial1Done THEN
				tonTimeOut(IN:= FALSE);
				G_Robot.RobotKukaCmd.bRobotPalletFiducial1 := FALSE;
				arrStepUsedTime[1] := tonStepTimer.ET;
				tonStepTimer(IN:=FALSE);
				iStep := 40;
			ELSIF tonTimeOut.Q THEN
				tonTimeOut(IN:= FALSE);
				G_Robot.RobotKukaCmd.bRobotPalletFiducial1 := FALSE;
				G_Error.E20_RobotTimeOutFailToPalletFiducial_1 := TRUE;
				iStep := 10;
			END_IF
			
		40: //Vision capture pallet fiducial 1
			arrStepStatus[2] := 'Step 2: Trigger Vision Capture';
			tonStepTimer(IN:=TRUE, PT:=T#999999S);
			IF NOT G_MachineControl.stMachineOperateMode.DRYRUN THEN
				G_Vision.V20_bRespone := FALSE;
				G_Vision.V20_sSendCmd := 'TRG,0';
				G_Vision.V20_bTrigger := TRUE;		
			END_IF
			iStep := 50;
			
		
		50: //Waiting vision capture done
			tonTimeOut(IN:= TRUE,PT:= tTimeOut);
			IF G_Vision.V20_bRespone OR G_MachineControl.stMachineOperateMode.DRYRUN THEN
				tonTimeOut(IN:= FALSE);
				G_Vision.V20_bTrigger := FALSE;
				arrStepUsedTime[2] := tonStepTimer.ET;
				tonStepTimer(IN:=FALSE);
				iStep := 60;
			ELSIF tonTimeOut.Q THEN
				tonTimeOut(IN:= FALSE);
				G_Vision.V20_bTrigger := FALSE;	
				G_Error.E20_VisionTimeOutInspection	:= TRUE;
				iStep := 40;
			END_IF
			
		60:
			G_Robot.RobotKukaCmd.rRobotPlace_X := G_Values.VA20_stPalletPosition.stFiducialDistance2Value.Xpos;
			G_Robot.RobotKukaCmd.rRobotPlace_Y := G_Values.VA20_stPalletPosition.stFiducialDistance2Value.Ypos;
			G_Robot.RobotKukaCmd.rRobotPlace_Z := 0; //G_Values.VA20_stPalletPosition.stFiducialDistance2Value.Zpos;
			G_Robot.RobotKukaCmd.rRobotPlace_A := G_Values.VA20_stPalletPosition.stFiducialDistance2Value.Apos;
			iStep := 70;
			
		70: //Robot move to pallet fiducial 2
			arrStepStatus[3] := 'Step 3: Robot go to pallet fiducial 2';
			tonStepTimer(IN:=TRUE, PT:=T#999999S);
			G_Robot.RobotKukaCmd.bRobotPalletFiducial2 := TRUE;
			iStep := 80;
			
		80:
			IF NOT G_Robot.RobotKukaCmd.bRobotPalletFiducial2Done THEN
				iStep := 90;
			END_IF
			
		90: //Robot move pallet fiducial 2 done
			tonTimeOut(IN:= TRUE,PT:= tTimeOut);
			IF G_Robot.RobotKukaCmd.bRobotPalletFiducial2Done THEN
				tonTimeOut(IN:= FALSE);
				G_Robot.RobotKukaCmd.bRobotPalletFiducial2 := FALSE;
				arrStepUsedTime[3] := tonStepTimer.ET;
				tonStepTimer(IN:=FALSE);
				iStep := 100;
			ELSIF tonTimeOut.Q THEN
				tonTimeOut(IN:= FALSE);
				G_Robot.RobotKukaCmd.bRobotPalletFiducial2 := FALSE;
				G_Error.E20_RobotTimeOutFailToPalletFiducial_2 := TRUE;
				iStep := 60;
			END_IF
			
		100: //Vision capture pallet fiducial 2
			arrStepStatus[4] := 'Step 4: Trigger Vision Capture';
			tonStepTimer(IN:=TRUE, PT:=T#999999S);
			IF NOT G_MachineControl.stMachineOperateMode.DRYRUN THEN
				G_Vision.V20_bRespone := FALSE;
				G_Vision.V20_sSendCmd := 'TRG,1';
				G_Vision.V20_bTrigger := TRUE;	
			END_IF			
			iStep := 110;
		
		110: //Waiting vision capture done
			tonTimeOut(IN:= TRUE,PT:= tTimeOut);
			IF G_Vision.V20_bRespone OR G_MachineControl.stMachineOperateMode.DRYRUN THEN
				tonTimeOut(IN:= FALSE);
				G_Vision.V20_bTrigger := FALSE;
				arrStepUsedTime[4] := tonStepTimer.ET;
				tonStepTimer(IN:=FALSE);
				iStep := 120;
			ELSIF tonTimeOut.Q THEN
				tonTimeOut(IN:= FALSE);
				G_Vision.V20_bTrigger := FALSE;	
				G_Error.E20_VisionTimeOutInspection	:= TRUE;
				iStep := 100;
			END_IF
			
		120: //Waiting Tray Ready
			arrStepStatus[5] := 'Step 5: Waiting Tray Ready';
			tonStepTimer(IN:=TRUE, PT:=T#999999S);
			IF bStart AND NOT G_MachineControl.arrstStationControl[2].bByPassStation AND G_Auto.A20_bMESCheckDone AND G_Auto.A20_bMESPass 
				AND NOT G_MachineControl.arrstStationControl[2].bJobDone AND G_Auto.A20_bTrayReady THEN
				arrStepUsedTime[5] := tonStepTimer.ET;
				tonStepTimer(IN:=FALSE);
				iStep := 130;	
			ELSIF bStart AND NOT G_MachineControl.arrstStationControl[2].bByPassStation AND G_Auto.A20_bMESCheckDone AND G_Auto.A20_bMESPass 
				AND NOT G_MachineControl.arrstStationControl[2].bJobDone AND NOT G_Auto.A20_bTrayReady AND NOT G_Auto.A20_bRobotAtStandbyTray THEN
				iStep := 2000; //go to standby at tray
			END_IF
			
		130: //Robot move to tray fiducial 1
			arrStepStatus[6] := 'Step 6: Robot go to tray fiducial 1';
			tonStepTimer(IN:=TRUE, PT:=T#999999S);
			G_Auto.A20_bRobotAtStandbyTray := FALSE;
			G_Robot.RobotKukaCmd.bRobotTrayFiducial1 := TRUE;
			iStep := 140; 
			
		140:
			IF NOT G_Robot.RobotKukaCmd.bRobotTrayFiducial1Done THEN
				iStep := 150;
			END_IF
			
		150://Robot move tray fiducial 1 done
			tonTimeOut(IN:= TRUE,PT:= tTimeOut);
			IF G_Robot.RobotKukaCmd.bRobotTrayFiducial1Done THEN
				tonTimeOut(IN:= FALSE);
				G_Robot.RobotKukaCmd.bRobotTrayFiducial1 := FALSE;
				arrStepUsedTime[6] := tonStepTimer.ET;
				tonStepTimer(IN:=FALSE);
				iStep := 160;
			ELSIF tonTimeOut.Q THEN
				tonTimeOut(IN:= FALSE);
				G_Robot.RobotKukaCmd.bRobotTrayFiducial1 := FALSE;
				G_Error.E20_RobotTimeOutFailToTrayFiducial_1 := TRUE;
				iStep := 120;
			END_IF
			
